// TwinCAT 3 PLC project Main
// ProgramVersion: 3.1.4024.0
// libraries:
//   Tc2_Standard, * (Beckhoff Automation GmbH)
//   Tc2_System, * (Beckhoff Automation GmbH)
//   Tc3_Module, * (Beckhoff Automation GmbH)
//   Tc3_Vision, * (Beckhoff Automation GmbH)
//   TcUnit, * (www.tcunit.org)
//   mobject-core,0.1.0,mobject
//   mobject-vision-nodepack,0.1.0,mobject
// project tree:
//   / PlcTask.TcTTO
//   POUs/ MAIN.TcPOU
//   Tests/Enums/ _ETcVn2dCodeSearchStrategy_TestSuite.TcPOU, _ETcVnAdaptiveThresholdMethod_TestSuite.TcPOU, _ETcVnBarcodeSearchDirection_TestSuite.TcPOU, _ETcVnBarcodeType_TestSuite.TcPOU, _ETcVnBlobCombination_TestSuite.TcPOU, _ETcVnBorderInterpolationMethod_TestSuite.TcPOU, _ETcVnColorSpaceTransform_TestSuite.TcPOU
// real-time tasks:
//   TASK PlcTask: cycle T#10ms, priority 20, ADS port 350

CONFIGURATION Main
    RESOURCE PLC ON TwinCAT3
        TASK PlcTask(INTERVAL := T#10ms, PRIORITY := 20);
        PROGRAM MAIN WITH PlcTask : MAIN;
    END_RESOURCE
END_CONFIGURATION

// ---- POUs/MAIN.TcPOU
PROGRAM MAIN
VAR
	
    // enums
    _ETcVn2dCodeSearchStrategy_TestSuite : _ETcVn2dCodeSearchStrategy_TestSuite;
    _ETcVnAdaptiveThresholdMethod_TestSuite : _ETcVnAdaptiveThresholdMethod_TestSuite;
    _ETcVnBarcodeSearchDirection_TestSuite : _ETcVnBarcodeSearchDirection_TestSuite;
    _ETcVnBarcodeType_TestSuite : _ETcVnBarcodeType_TestSuite;
    _ETcVnBlobCombination_TestSuite : _ETcVnBlobCombination_TestSuite;
    _ETcVnBorderInterpolationMethod_TestSuite : _ETcVnBorderInterpolationMethod_TestSuite;
    //_ETcVnCalibrationPattern_TestSuite : _ETcVnCalibrationPattern_TestSuite;
    //_ETcVnCalibrationPatternOrigin_TestSuite : _ETcVnCalibrationPatternOrigin_TestSuite;
    //_ETcVnCameraState_TestSuite : _ETcVnCameraState_TestSuite;
    //_ETcVnClusteringAlgorithm_TestSuite : _ETcVnClusteringAlgorithm_TestSuite;
    //_ETcVnColorMap_TestSuite : _ETcVnColorMap_TestSuite;
    //_ETcVnColorMapSize_TestSuite : _ETcVnColorMapSize_TestSuite;
    _ETcVnColorSpaceTransform_TestSuite : _ETcVnColorSpaceTransform_TestSuite;
    //_ETcVnColorTrainingMethod_TestSuite : _ETcVnColorTrainingMethod_TestSuite;
    //_ETcVnConnectedComponentsAlgorithm_TestSuite : _ETcVnConnectedComponentsAlgorithm_TestSuite;
    //_ETcVnContainerExportFormat_TestSuite : _ETcVnContainerExportFormat_TestSuite;
    //_ETcVnContourApproximationMethod_TestSuite : _ETcVnContourApproximationMethod_TestSuite;
    //_ETcVnContourRetrievalMode_TestSuite : _ETcVnContourRetrievalMode_TestSuite;
    //_ETcVnContoursMatchComparisonMethod_TestSuite : _ETcVnContoursMatchComparisonMethod_TestSuite;
    //_ETcVnDiffusivityTypeKAZE_TestSuite : _ETcVnDiffusivityTypeKAZE_TestSuite;
    //_ETcVnDistanceTransformationLabel_TestSuite : _ETcVnDistanceTransformationLabel_TestSuite;
    //_ETcVnDistanceTransformationMask_TestSuite : _ETcVnDistanceTransformationMask_TestSuite;
    //_ETcVnDistanceType_TestSuite : _ETcVnDistanceType_TestSuite;
    //_ETcVnDrawMatchesFlags_TestSuite : _ETcVnDrawMatchesFlags_TestSuite;
    //_ETcVnDrawShape_TestSuite : _ETcVnDrawShape_TestSuite;
    //_ETcVnEdgeDetectionAlgorithm_TestSuite : _ETcVnEdgeDetectionAlgorithm_TestSuite;
    //_ETcVnEdgeDirection_TestSuite : _ETcVnEdgeDirection_TestSuite;
    //_ETcVnElementType_TestSuite : _ETcVnElementType_TestSuite;
    //_ETcVnEstimationAlgorithm_TestSuite : _ETcVnEstimationAlgorithm_TestSuite;
    //_ETcVnExtremePointDirection_TestSuite : _ETcVnExtremePointDirection_TestSuite;
    //_ETcVnFeatureDescriptorTypeAKAZE_TestSuite : _ETcVnFeatureDescriptorTypeAKAZE_TestSuite;
    //_ETcVnFeatureScalingType_TestSuite : _ETcVnFeatureScalingType_TestSuite;
    //_ETcVnFeatureScoreTypeORB_TestSuite : _ETcVnFeatureScoreTypeORB_TestSuite;
    //_ETcVnFilterDirection_TestSuite : _ETcVnFilterDirection_TestSuite;
    //_ETcVnFlipAxis_TestSuite : _ETcVnFlipAxis_TestSuite;
    //_ETcVnFontType_TestSuite : _ETcVnFontType_TestSuite;
    //_ETcVnHoughMethod_TestSuite : _ETcVnHoughMethod_TestSuite;
    //_ETcVnInitializableFunction_TestSuite : _ETcVnInitializableFunction_TestSuite;
    //_ETcVnInterpolationType_TestSuite : _ETcVnInterpolationType_TestSuite;
    //_ETcVnKeypointDetectionTypeAGAST_TestSuite : _ETcVnKeypointDetectionTypeAGAST_TestSuite;
    //_ETcVnKeypointDetectionTypeFAST_TestSuite : _ETcVnKeypointDetectionTypeFAST_TestSuite;
    //_ETcVnKnn_TestSuite : _ETcVnKnn_TestSuite;
    //_ETcVnLineType_TestSuite : _ETcVnLineType_TestSuite;
    //_ETcVnMorphologicalOperator_TestSuite : _ETcVnMorphologicalOperator_TestSuite;
    //_ETcVnNbc_TestSuite : _ETcVnNbc_TestSuite;
    //_ETcVnNormalizationType_TestSuite : _ETcVnNormalizationType_TestSuite;
    //_ETcVnOcrModelType_TestSuite : _ETcVnOcrModelType_TestSuite;
    //_ETcVnOcrOptions_TestSuite : _ETcVnOcrOptions_TestSuite;
    //_ETcVnOrientationMethod_TestSuite : _ETcVnOrientationMethod_TestSuite;
    //_ETcVnPaddingMode_TestSuite : _ETcVnPaddingMode_TestSuite;
    //_ETcVnPixelConnectivity_TestSuite : _ETcVnPixelConnectivity_TestSuite;
    //_ETcVnPixelEncoding_TestSuite : _ETcVnPixelEncoding_TestSuite;
    //_ETcVnPixelPackMode_TestSuite : _ETcVnPixelPackMode_TestSuite;
    //_ETcVnPrototypeClusterer_TestSuite : _ETcVnPrototypeClusterer_TestSuite;
    //_ETcVnRectangleIntersection_TestSuite : _ETcVnRectangleIntersection_TestSuite;
    //_ETcVnRotationAngle_TestSuite : _ETcVnRotationAngle_TestSuite;
    //_ETcVnRTrees_TestSuite : _ETcVnRTrees_TestSuite;
    //_ETcVnSignedNormalization_TestSuite : _ETcVnSignedNormalization_TestSuite;
    //_ETcVnSolvePnPMethod_TestSuite : _ETcVnSolvePnPMethod_TestSuite;
    //_ETcVnSta_TestSuite : _ETcVnSta_TestSuite;
    //_ETcVnStructuringElementShape_TestSuite : _ETcVnStructuringElementShape_TestSuite;
    //_ETcVnSvm_TestSuite : _ETcVnSvm_TestSuite;
    //_ETcVnSvmKernelType_TestSuite : _ETcVnSvmKernelType_TestSuite;
    //_ETcVnSvmSgdClassifierMarginType_TestSuite : _ETcVnSvmSgdClassifierMarginType_TestSuite;
    //_ETcVnSvmSgdClassifierType_TestSuite : _ETcVnSvmSgdClassifierType_TestSuite;
    //_ETcVnTemplateMatchMethod_TestSuite : _ETcVnTemplateMatchMethod_TestSuite;
    //_ETcVnThresholdType_TestSuite : _ETcVnThresholdType_TestSuite;
    //_ETcVnVectorCompareMethod_TestSuite : _ETcVnVectorCompareMethod_TestSuite;
    //_ETcVnWorldCoordinateSystem_TestSuite : _ETcVnWorldCoordinateSystem_TestSuite;
    //_ETcWatchdogAccumulationType_TestSuite : _ETcWatchdogAccumulationType_TestSuite;
    //_GEV_CAMERA_STATE_TestSuite : _GEV_CAMERA_STATE_TestSuite;
    
    //structs
	
END_VAR

END_PROGRAM

// ---- Tests/Enums/_ETcVn2dCodeSearchStrategy_TestSuite.TcPOU
FUNCTION_BLOCK _ETcVn2dCodeSearchStrategy_TestSuite EXTENDS TcUnit.FB_TestSuite
VAR
END_VAR

TestAddress();
TestClearReference();
TestClone();
TestTypeNameReturnsExpected();
TestIdentifierReturnsExpected();
TestMakeReferenceToFollowsReference();
TestMakeReferenceToUpdatesReference();
TestSize();
TestValueReturnsExpectedAfterInit();
TestValueReturnsExpectedAfterChange();
TestSerializeTypeWith();
TestSerializeWith();
TestTryDeserializeFrom();
TestTryMakeReferenceToFollowsReference();
TestTryMakeReferenceToUpdatesReference();

METHOD PUBLIC TestAddress
VAR
    _type : _ETcVn2dCodeSearchStrategy(ETcVn2dCodeSearchStrategy.TCVN_CSS_DEFAULT);
    notExpected : PVOID := 0;
    actual : PVOID;
END_VAR
TEST('TestAddress');

actual := _type.Address;

AssertFalse(
    Condition := (notExpected = actual),
    Message := 'Type did not return a valid address.'
);

TEST_FINISHED();
END_METHOD

METHOD PUBLIC TestClearReference
VAR
    _type : _ETcVn2dCodeSearchStrategy(ETcVn2dCodeSearchStrategy.TCVN_CSS_DEFAULT);
	target : ETcVn2dCodeSearchStrategy := ETcVn2dCodeSearchStrategy.TCVN_CSS_DEFAULT;
    expected : ETcVn2dCodeSearchStrategy := ETcVn2dCodeSearchStrategy.TCVN_CSS_DEFAULT;
    actual : ETcVn2dCodeSearchStrategy;
END_VAR
TEST('TestClearReference');

_type.MakeReferenceTo(target);
_type.ClearReference();
target := ETcVn2dCodeSearchStrategy.TCVN_CSS_FIRST_FLIPPED;

actual := _type.Value;

AssertEquals(
    Expected := expected,
    Actual := actual,
    Message := 'Value continued to follow target.'
);

TEST_FINISHED();
END_METHOD

METHOD PUBLIC TestClone
VAR
    _type : _ETcVn2dCodeSearchStrategy(ETcVn2dCodeSearchStrategy.TCVN_CSS_DEFAULT);
	clone : I_Datatype;
	isValidClone : BOOL;
	compareResult : DINT;
END_VAR
TEST('TestClone');

clone := _type.Clone();

isValidClone := clone <> 0;

IF isValidClone THEN
	compareResult := memcmp(_type.Address, clone.Address, clone.Size);
END_IF

AssertTrue(
	Condition := isValidClone,
	Message := 'Clone did not produce a clone'
);

AssertEquals_DINT(
	Expected := 0,
    Actual := compareResult,
    Message := 'Clone did not return a valid clone.'
);

clone.Dispose();

TEST_FINISHED();
END_METHOD

METHOD PUBLIC TestIdentifierReturnsExpected
VAR
    _type : _ETcVn2dCodeSearchStrategy(ETcVn2dCodeSearchStrategy.TCVN_CSS_DEFAULT);
    expected : STRING := 'ETcVn2dCodeSearchStrategy';
    actual : STRING;
END_VAR
TEST('TestIdentifierReturnsExpected');

actual := _type.Identifier;

AssertEquals_STRING(
    Expected := expected,
    Actual := actual,
    Message := 'Type did not return correct iec type.'
);

TEST_FINISHED();
END_METHOD

METHOD PUBLIC TestMakeReferenceToFollowsReference
VAR
    _type : _ETcVn2dCodeSearchStrategy(ETcVn2dCodeSearchStrategy.TCVN_CSS_DEFAULT);
	target : ETcVn2dCodeSearchStrategy := ETcVn2dCodeSearchStrategy.TCVN_CSS_DEFAULT;
    expected : ETcVn2dCodeSearchStrategy := ETcVn2dCodeSearchStrategy.TCVN_CSS_FIRST_FLIPPED;
    actual : ETcVn2dCodeSearchStrategy;
END_VAR
TEST('TestMakeReferenceToFollowsReference');

_type.MakeReferenceTo(target);
target := ETcVn2dCodeSearchStrategy.TCVN_CSS_FIRST_FLIPPED;

actual := _type.Value;

AssertEquals(
    Expected := expected,
    Actual := actual,
    Message := 'Value did not follow target change.'
);

TEST_FINISHED();
END_METHOD

METHOD PUBLIC TestMakeReferenceToUpdatesReference
VAR
    _type : _ETcVn2dCodeSearchStrategy(ETcVn2dCodeSearchStrategy.TCVN_CSS_DEFAULT);
	target : ETcVn2dCodeSearchStrategy := ETcVn2dCodeSearchStrategy.TCVN_CSS_DEFAULT;
    expected : ETcVn2dCodeSearchStrategy := ETcVn2dCodeSearchStrategy.TCVN_CSS_FIRST_FLIPPED;
    actual : ETcVn2dCodeSearchStrategy;
END_VAR
TEST('TestMakeReferenceToUpdatesReference');

_type.MakeReferenceTo(target);
_type.Value := ETcVn2dCodeSearchStrategy.TCVN_CSS_FIRST_FLIPPED;

actual := target;

AssertEquals(
    Expected := expected,
    Actual := actual,
    Message := 'Value did not update target.'
);

TEST_FINISHED();
END_METHOD

METHOD PUBLIC TestSerializeTypeWith
VAR
    _type : _ETcVn2dCodeSearchStrategy(ETcVn2dCodeSearchStrategy.TCVN_CSS_DEFAULT);
    serializer : JsonSerializer;
    expected : STRING(500) := '{"typeName":"ENUM","identifier":"ETcVn2dCodeSearchStrategy","enumerations":["TCVN_CSS_DEFAULT","TCVN_CSS_FIRST_FLIPPED","TCVN_CSS_FIRST_INVERTED","TCVN_CSS_FIRST_NOT_FLIPPED","TCVN_CSS_FIRST_NOT_INVERTED","TCVN_CSS_ONLY_FLIPPED","TCVN_CSS_ONLY_INVERTED","TCVN_CSS_ONLY_NOT_FLIPPED","TCVN_CSS_ONLY_NOT_INVERTED"],"baseType":{"typeName":"UDINT","minValue":0,"maxValue":4294967295,"isSigned":false,"isFloat":false}}';
    actual : STRING(500);
END_VAR
TEST('TestSerializeTypeWith');

serializer.Reset();
_type.SerializeTypeWith(serializer);
serializer.TryGetSerializedData(ADR(actual), SIZEOF(actual));

AssertEquals_STRING(
    Expected := expected,
    Actual := actual,
    Message := 'Serialization of type did not return correct string.'
);

TEST_FINISHED();
END_METHOD

METHOD PUBLIC TestSerializeWith
VAR
    _type : _ETcVn2dCodeSearchStrategy(ETcVn2dCodeSearchStrategy.TCVN_CSS_DEFAULT);
    serializer : JsonSerializer;
    expected : STRING := '"TCVN_CSS_DEFAULT"';
    actual : STRING(500);
END_VAR
TEST('TestSerializeWith');

serializer.Reset();
_type.SerializeWith(serializer);
serializer.TryGetSerializedData(ADR(actual), SIZEOF(actual));

AssertEquals_STRING(
    Expected := expected,
    Actual := actual,
    Message := 'Serialization of type data did not return correct string.'
);

TEST_FINISHED();
END_METHOD

METHOD PUBLIC TestSize
VAR
    _type : _ETcVn2dCodeSearchStrategy(ETcVn2dCodeSearchStrategy.TCVN_CSS_DEFAULT);
    expected : UDINT := SIZEOF(ETcVn2dCodeSearchStrategy);
    actual : UDINT;
END_VAR
TEST('TestSize');

actual := _type.Size;

AssertEquals_UDINT(
    Expected := Expected,
    Actual := actual,
    Message := 'Type did not return the correct size.'
);

TEST_FINISHED();
END_METHOD

METHOD PUBLIC TestTryDeserializeFrom
VAR
    deserializer : JsonDeserializer;
    feedback : DeserializerFeedback;
    json : STRING := '"TCVN_CSS_DEFAULT"';
    _type : _ETcVn2dCodeSearchStrategy(ETcVn2dCodeSearchStrategy.TCVN_CSS_DEFAULT);
    expected : ETcVn2dCodeSearchStrategy := ETcVn2dCodeSearchStrategy.TCVN_CSS_DEFAULT;
    actual : ETcVn2dCodeSearchStrategy;
 END_VAR
TEST('TestTryDeserializeFrom');

deserializer.Reset();
deserializer.TryLoad(json);
_type.TryDeserializeFrom(Deserializer, Feedback);

actual := _type.Value;

AssertEquals(
    Expected := expected,
    Actual := actual,
    Message := 'Type did not deserialize correctly.'
);

TEST_FINISHED();
END_METHOD

METHOD PUBLIC TestTryMakeReferenceToFollowsReference
VAR
    _type : _ETcVn2dCodeSearchStrategy(ETcVn2dCodeSearchStrategy.TCVN_CSS_DEFAULT);
	target : _ETcVn2dCodeSearchStrategy(ETcVn2dCodeSearchStrategy.TCVN_CSS_DEFAULT);
    expected : ETcVn2dCodeSearchStrategy := ETcVn2dCodeSearchStrategy.TCVN_CSS_FIRST_FLIPPED;
    actual : ETcVn2dCodeSearchStrategy;
END_VAR
TEST('TestTryMakeReferenceToFollowsReference');

_type.TryMakeReferenceTo(target);
target.Value := ETcVn2dCodeSearchStrategy.TCVN_CSS_FIRST_FLIPPED;

actual := _type.Value;

AssertEquals(
    Expected := expected,
    Actual := actual,
    Message := 'Value did not follow target change.'
);

TEST_FINISHED();
END_METHOD

METHOD PUBLIC TestTryMakeReferenceToUpdatesReference
VAR
    _type : _ETcVn2dCodeSearchStrategy(ETcVn2dCodeSearchStrategy.TCVN_CSS_DEFAULT);
	target : _ETcVn2dCodeSearchStrategy(ETcVn2dCodeSearchStrategy.TCVN_CSS_DEFAULT);
    expected : ETcVn2dCodeSearchStrategy := ETcVn2dCodeSearchStrategy.TCVN_CSS_FIRST_FLIPPED;
    actual : ETcVn2dCodeSearchStrategy;
END_VAR
TEST('TestTryMakeReferenceToUpdatesReference');

_type.TryMakeReferenceTo(target);
_type.Value := ETcVn2dCodeSearchStrategy.TCVN_CSS_FIRST_FLIPPED;

actual := target.Value;

AssertEquals(
    Expected := expected,
    Actual := actual,
    Message := 'Value did not update target.'
);

TEST_FINISHED();
END_METHOD

METHOD PUBLIC TestTypeNameReturnsExpected
VAR
    _type : _ETcVn2dCodeSearchStrategy(ETcVn2dCodeSearchStrategy.TCVN_CSS_DEFAULT);
    expected : STRING := 'ENUM';
    actual : STRING;
END_VAR
TEST('TestTypeNameReturnsExpected');

actual := _type.TypeName;

AssertEquals_STRING(
    Expected := expected,
    Actual := actual,
    Message := 'Type did not return correct iec type.'
);

TEST_FINISHED();
END_METHOD

METHOD PUBLIC TestValueReturnsExpectedAfterChange
VAR
    _type : _ETcVn2dCodeSearchStrategy(ETcVn2dCodeSearchStrategy.TCVN_CSS_DEFAULT);
    expected : ETcVn2dCodeSearchStrategy := ETcVn2dCodeSearchStrategy.TCVN_CSS_FIRST_FLIPPED;
    actual : ETcVn2dCodeSearchStrategy;
END_VAR
TEST('TestValueReturnsExpectedAfterChange');

_type.Value := ETcVn2dCodeSearchStrategy.TCVN_CSS_FIRST_FLIPPED;

actual := _type.Value;

AssertEquals(
    Expected := expected,
    Actual := actual,
    Message := 'Expected value not returned after change.'
);

TEST_FINISHED();
END_METHOD

METHOD PUBLIC TestValueReturnsExpectedAfterInit
VAR
    _type : _ETcVn2dCodeSearchStrategy(ETcVn2dCodeSearchStrategy.TCVN_CSS_DEFAULT);
    expected : ETcVn2dCodeSearchStrategy := ETcVn2dCodeSearchStrategy.TCVN_CSS_DEFAULT;
    actual : ETcVn2dCodeSearchStrategy;
END_VAR
TEST('TestValueReturnsExpectedAfterInit');

actual := _type.Value;

AssertEquals(
    Expected := expected,
    Actual := actual,
    Message := 'Expected value not returned after Init.'
);

TEST_FINISHED();
END_METHOD

END_FUNCTION_BLOCK

// ---- Tests/Enums/_ETcVnAdaptiveThresholdMethod_TestSuite.TcPOU
FUNCTION_BLOCK _ETcVnAdaptiveThresholdMethod_TestSuite EXTENDS TcUnit.FB_TestSuite
VAR
END_VAR

TestAddress();
TestClearReference();
TestClone();
TestTypeNameReturnsExpected();
TestIdentifierReturnsExpected();
TestMakeReferenceToFollowsReference();
TestMakeReferenceToUpdatesReference();
TestSize();
TestValueReturnsExpectedAfterInit();
TestValueReturnsExpectedAfterChange();
TestSerializeTypeWith();
TestSerializeWith();
TestTryDeserializeFrom();
TestTryMakeReferenceToFollowsReference();
TestTryMakeReferenceToUpdatesReference();

METHOD PUBLIC TestAddress
VAR
    _type : _ETcVnAdaptiveThresholdMethod(ETcVnAdaptiveThresholdMethod.TCVN_ATM_MEAN);
    notExpected : PVOID := 0;
    actual : PVOID;
END_VAR
TEST('TestAddress');

actual := _type.Address;

AssertFalse(
    Condition := (notExpected = actual),
    Message := 'Type did not return a valid address.'
);

TEST_FINISHED();
END_METHOD

METHOD PUBLIC TestClearReference
VAR
    _type : _ETcVnAdaptiveThresholdMethod(ETcVnAdaptiveThresholdMethod.TCVN_ATM_MEAN);
	target : ETcVnAdaptiveThresholdMethod := ETcVnAdaptiveThresholdMethod.TCVN_ATM_MEAN;
    expected : ETcVnAdaptiveThresholdMethod := ETcVnAdaptiveThresholdMethod.TCVN_ATM_MEAN;
    actual : ETcVnAdaptiveThresholdMethod;
END_VAR
TEST('TestClearReference');

_type.MakeReferenceTo(target);
_type.ClearReference();
target := ETcVnAdaptiveThresholdMethod.TCVN_ATM_GAUSSIAN;

actual := _type.Value;

AssertEquals(
    Expected := expected,
    Actual := actual,
    Message := 'Value continued to follow target.'
);

TEST_FINISHED();
END_METHOD

METHOD PUBLIC TestClone
VAR
    _type : _ETcVnAdaptiveThresholdMethod(ETcVnAdaptiveThresholdMethod.TCVN_ATM_MEAN);
	clone : I_Datatype;
	isValidClone : BOOL;
	compareResult : DINT;
END_VAR
TEST('TestClone');

clone := _type.Clone();

isValidClone := clone <> 0;

IF isValidClone THEN
	compareResult := memcmp(_type.Address, clone.Address, clone.Size);
END_IF

AssertTrue(
	Condition := isValidClone,
	Message := 'Clone did not produce a clone'
);

AssertEquals_DINT(
	Expected := 0,
    Actual := compareResult,
    Message := 'Clone did not return a valid clone.'
);

clone.Dispose();

TEST_FINISHED();
END_METHOD

METHOD PUBLIC TestIdentifierReturnsExpected
VAR
    _type : _ETcVnAdaptiveThresholdMethod(ETcVnAdaptiveThresholdMethod.TCVN_ATM_MEAN);
    expected : STRING := 'ETcVnAdaptiveThresholdMethod';
    actual : STRING;
END_VAR
TEST('TestIdentifierReturnsExpected');

actual := _type.Identifier;

AssertEquals_STRING(
    Expected := expected,
    Actual := actual,
    Message := 'Type did not return correct iec type.'
);

TEST_FINISHED();
END_METHOD

METHOD PUBLIC TestMakeReferenceToFollowsReference
VAR
    _type : _ETcVnAdaptiveThresholdMethod(ETcVnAdaptiveThresholdMethod.TCVN_ATM_MEAN);
	target : ETcVnAdaptiveThresholdMethod := ETcVnAdaptiveThresholdMethod.TCVN_ATM_MEAN;
    expected : ETcVnAdaptiveThresholdMethod := ETcVnAdaptiveThresholdMethod.TCVN_ATM_GAUSSIAN;
    actual : ETcVnAdaptiveThresholdMethod;
END_VAR
TEST('TestMakeReferenceToFollowsReference');

_type.MakeReferenceTo(target);
target := ETcVnAdaptiveThresholdMethod.TCVN_ATM_GAUSSIAN;

actual := _type.Value;

AssertEquals(
    Expected := expected,
    Actual := actual,
    Message := 'Value did not follow target change.'
);

TEST_FINISHED();
END_METHOD

METHOD PUBLIC TestMakeReferenceToUpdatesReference
VAR
    _type : _ETcVnAdaptiveThresholdMethod(ETcVnAdaptiveThresholdMethod.TCVN_ATM_MEAN);
	target : ETcVnAdaptiveThresholdMethod := ETcVnAdaptiveThresholdMethod.TCVN_ATM_MEAN;
    expected : ETcVnAdaptiveThresholdMethod := ETcVnAdaptiveThresholdMethod.TCVN_ATM_GAUSSIAN;
    actual : ETcVnAdaptiveThresholdMethod;
END_VAR
TEST('TestMakeReferenceToUpdatesReference');

_type.MakeReferenceTo(target);
_type.Value := ETcVnAdaptiveThresholdMethod.TCVN_ATM_GAUSSIAN;

actual := target;

AssertEquals(
    Expected := expected,
    Actual := actual,
    Message := 'Value did not update target.'
);

TEST_FINISHED();
END_METHOD

METHOD PUBLIC TestSerializeTypeWith
VAR
    _type : _ETcVnAdaptiveThresholdMethod(ETcVnAdaptiveThresholdMethod.TCVN_ATM_MEAN);
    serializer : JsonSerializer;
    expected : STRING(500) := '{"typeName":"ENUM","identifier":"ETcVnAdaptiveThresholdMethod","enumerations":["TCVN_ATM_MEAN","TCVN_ATM_GAUSSIAN"],"baseType":{"typeName":"DINT","minValue":-2147483648,"maxValue":2147483647,"isSigned":true,"isFloat":false}}'; 
    actual : STRING(500);
END_VAR
TEST('TestSerializeTypeWith');

serializer.Reset();
_type.SerializeTypeWith(serializer);
serializer.TryGetSerializedData(ADR(actual), SIZEOF(actual));

AssertEquals_STRING(
    Expected := expected,
    Actual := actual,
    Message := 'Serialization of type did not return correct string.'
);

TEST_FINISHED();
END_METHOD

METHOD PUBLIC TestSerializeWith
VAR
    _type : _ETcVnAdaptiveThresholdMethod(ETcVnAdaptiveThresholdMethod.TCVN_ATM_MEAN);
    serializer : JsonSerializer;
    expected : STRING := '"TCVN_ATM_MEAN"';
    actual : STRING(500);
END_VAR
TEST('TestSerializeWith');

serializer.Reset();
_type.SerializeWith(serializer);
serializer.TryGetSerializedData(ADR(actual), SIZEOF(actual));

AssertEquals_STRING(
    Expected := expected,
    Actual := actual,
    Message := 'Serialization of type data did not return correct string.'
);

TEST_FINISHED();
END_METHOD

METHOD PUBLIC TestSize
VAR
    _type : _ETcVnAdaptiveThresholdMethod(ETcVnAdaptiveThresholdMethod.TCVN_ATM_MEAN);
    expected : UDINT := SIZEOF(ETcVnAdaptiveThresholdMethod);
    actual : UDINT;
END_VAR
TEST('TestSize');

actual := _type.Size;

AssertEquals_UDINT(
    Expected := Expected,
    Actual := actual,
    Message := 'Type did not return the correct size.'
);

TEST_FINISHED();
END_METHOD

METHOD PUBLIC TestTryDeserializeFrom
VAR
    deserializer : JsonDeserializer;
    feedback : DeserializerFeedback;
    json : STRING := '"TCVN_ATM_MEAN"';
    _type : _ETcVnAdaptiveThresholdMethod(ETcVnAdaptiveThresholdMethod.TCVN_ATM_MEAN);
    expected : ETcVnAdaptiveThresholdMethod := ETcVnAdaptiveThresholdMethod.TCVN_ATM_MEAN;
    actual : ETcVnAdaptiveThresholdMethod;
 END_VAR
TEST('TestTryDeserializeFrom');

deserializer.Reset();
deserializer.TryLoad(json);
_type.TryDeserializeFrom(Deserializer, Feedback);

actual := _type.Value;

AssertEquals(
    Expected := expected,
    Actual := actual,
    Message := 'Type did not deserialize correctly.'
);

TEST_FINISHED();
END_METHOD

METHOD PUBLIC TestTryMakeReferenceToFollowsReference
VAR
    _type : _ETcVnAdaptiveThresholdMethod(ETcVnAdaptiveThresholdMethod.TCVN_ATM_MEAN);
	target : _ETcVnAdaptiveThresholdMethod(ETcVnAdaptiveThresholdMethod.TCVN_ATM_MEAN);
    expected : ETcVnAdaptiveThresholdMethod := ETcVnAdaptiveThresholdMethod.TCVN_ATM_GAUSSIAN;
    actual : ETcVnAdaptiveThresholdMethod;
END_VAR
TEST('TestTryMakeReferenceToFollowsReference');

_type.TryMakeReferenceTo(target);
target.Value := ETcVnAdaptiveThresholdMethod.TCVN_ATM_GAUSSIAN;

actual := _type.Value;

AssertEquals(
    Expected := expected,
    Actual := actual,
    Message := 'Value did not follow target change.'
);

TEST_FINISHED();
END_METHOD

METHOD PUBLIC TestTryMakeReferenceToUpdatesReference
VAR
    _type : _ETcVnAdaptiveThresholdMethod(ETcVnAdaptiveThresholdMethod.TCVN_ATM_MEAN);
	target : _ETcVnAdaptiveThresholdMethod(ETcVnAdaptiveThresholdMethod.TCVN_ATM_MEAN);
    expected : ETcVnAdaptiveThresholdMethod := ETcVnAdaptiveThresholdMethod.TCVN_ATM_GAUSSIAN;
    actual : ETcVnAdaptiveThresholdMethod;
END_VAR
TEST('TestTryMakeReferenceToUpdatesReference');

_type.TryMakeReferenceTo(target);
_type.Value := ETcVnAdaptiveThresholdMethod.TCVN_ATM_GAUSSIAN;

actual := target.Value;

AssertEquals(
    Expected := expected,
    Actual := actual,
    Message := 'Value did not update target.'
);

TEST_FINISHED();
END_METHOD

METHOD PUBLIC TestTypeNameReturnsExpected
VAR
    _type : _ETcVnAdaptiveThresholdMethod(ETcVnAdaptiveThresholdMethod.TCVN_ATM_MEAN);
    expected : STRING := 'ENUM';
    actual : STRING;
END_VAR
TEST('TestTypeNameReturnsExpected');

actual := _type.TypeName;

AssertEquals_STRING(
    Expected := expected,
    Actual := actual,
    Message := 'Type did not return correct iec type.'
);

TEST_FINISHED();
END_METHOD

METHOD PUBLIC TestValueReturnsExpectedAfterChange
VAR
    _type : _ETcVnAdaptiveThresholdMethod(ETcVnAdaptiveThresholdMethod.TCVN_ATM_MEAN);
    expected : ETcVnAdaptiveThresholdMethod := ETcVnAdaptiveThresholdMethod.TCVN_ATM_GAUSSIAN;
    actual : ETcVnAdaptiveThresholdMethod;
END_VAR
TEST('TestValueReturnsExpectedAfterChange');

_type.Value := ETcVnAdaptiveThresholdMethod.TCVN_ATM_GAUSSIAN;

actual := _type.Value;

AssertEquals(
    Expected := expected,
    Actual := actual,
    Message := 'Expected value not returned after change.'
);

TEST_FINISHED();
END_METHOD

METHOD PUBLIC TestValueReturnsExpectedAfterInit
VAR
    _type : _ETcVnAdaptiveThresholdMethod(ETcVnAdaptiveThresholdMethod.TCVN_ATM_MEAN);
    expected : ETcVnAdaptiveThresholdMethod := ETcVnAdaptiveThresholdMethod.TCVN_ATM_MEAN;
    actual : ETcVnAdaptiveThresholdMethod;
END_VAR
TEST('TestValueReturnsExpectedAfterInit');

actual := _type.Value;

AssertEquals(
    Expected := expected,
    Actual := actual,
    Message := 'Expected value not returned after Init.'
);

TEST_FINISHED();
END_METHOD

END_FUNCTION_BLOCK

// ---- Tests/Enums/_ETcVnBarcodeSearchDirection_TestSuite.TcPOU
FUNCTION_BLOCK _ETcVnBarcodeSearchDirection_TestSuite EXTENDS TcUnit.FB_TestSuite
VAR
END_VAR

TestAddress();
TestClearReference();
TestClone();
TestTypeNameReturnsExpected();
TestIdentifierReturnsExpected();
TestMakeReferenceToFollowsReference();
TestMakeReferenceToUpdatesReference();
TestSize();
TestValueReturnsExpectedAfterInit();
TestValueReturnsExpectedAfterChange();
TestSerializeTypeWith();
TestSerializeWith();
TestTryDeserializeFrom();
TestTryMakeReferenceToFollowsReference();
TestTryMakeReferenceToUpdatesReference();

METHOD PUBLIC TestAddress
VAR
    _type : _ETcVnBarcodeSearchDirection(ETcVnBarcodeSearchDirection.TCVN_BSD_ANY);
    notExpected : PVOID := 0;
    actual : PVOID;
END_VAR
TEST('TestAddress');

actual := _type.Address;

AssertFalse(
    Condition := (notExpected = actual),
    Message := 'Type did not return a valid address.'
);

TEST_FINISHED();
END_METHOD

METHOD PUBLIC TestClearReference
VAR
    _type : _ETcVnBarcodeSearchDirection(ETcVnBarcodeSearchDirection.TCVN_BSD_ANY);
	target : ETcVnBarcodeSearchDirection := ETcVnBarcodeSearchDirection.TCVN_BSD_ANY;
    expected : ETcVnBarcodeSearchDirection := ETcVnBarcodeSearchDirection.TCVN_BSD_ANY;
    actual : ETcVnBarcodeSearchDirection;
END_VAR
TEST('TestClearReference');

_type.MakeReferenceTo(target);
_type.ClearReference();
target := ETcVnBarcodeSearchDirection.TCVN_BSD_HORIZONTAL;

actual := _type.Value;

AssertEquals(
    Expected := expected,
    Actual := actual,
    Message := 'Value continued to follow target.'
);

TEST_FINISHED();
END_METHOD

METHOD PUBLIC TestClone
VAR
    _type : _ETcVnBarcodeSearchDirection(ETcVnBarcodeSearchDirection.TCVN_BSD_ANY);
	clone : I_Datatype;
	isValidClone : BOOL;
	compareResult : DINT;
END_VAR
TEST('TestClone');

clone := _type.Clone();

isValidClone := clone <> 0;

IF isValidClone THEN
	compareResult := memcmp(_type.Address, clone.Address, clone.Size);
END_IF

AssertTrue(
	Condition := isValidClone,
	Message := 'Clone did not produce a clone'
);

AssertEquals_DINT(
	Expected := 0,
    Actual := compareResult,
    Message := 'Clone did not return a valid clone.'
);

clone.Dispose();

TEST_FINISHED();
END_METHOD

METHOD PUBLIC TestIdentifierReturnsExpected
VAR
    _type : _ETcVnBarcodeSearchDirection(ETcVnBarcodeSearchDirection.TCVN_BSD_ANY);
    expected : STRING := 'ETcVnBarcodeSearchDirection';
    actual : STRING;
END_VAR
TEST('TestIdentifierReturnsExpected');

actual := _type.Identifier;

AssertEquals_STRING(
    Expected := expected,
    Actual := actual,
    Message := 'Type did not return correct iec type.'
);

TEST_FINISHED();
END_METHOD

METHOD PUBLIC TestMakeReferenceToFollowsReference
VAR
    _type : _ETcVnBarcodeSearchDirection(ETcVnBarcodeSearchDirection.TCVN_BSD_ANY);
	target : ETcVnBarcodeSearchDirection := ETcVnBarcodeSearchDirection.TCVN_BSD_ANY;
    expected : ETcVnBarcodeSearchDirection := ETcVnBarcodeSearchDirection.TCVN_BSD_HORIZONTAL;
    actual : ETcVnBarcodeSearchDirection;
END_VAR
TEST('TestMakeReferenceToFollowsReference');

_type.MakeReferenceTo(target);
target := ETcVnBarcodeSearchDirection.TCVN_BSD_HORIZONTAL;

actual := _type.Value;

AssertEquals(
    Expected := expected,
    Actual := actual,
    Message := 'Value did not follow target change.'
);

TEST_FINISHED();
END_METHOD

METHOD PUBLIC TestMakeReferenceToUpdatesReference
VAR
    _type : _ETcVnBarcodeSearchDirection(ETcVnBarcodeSearchDirection.TCVN_BSD_ANY);
	target : ETcVnBarcodeSearchDirection := ETcVnBarcodeSearchDirection.TCVN_BSD_ANY;
    expected : ETcVnBarcodeSearchDirection := ETcVnBarcodeSearchDirection.TCVN_BSD_HORIZONTAL;
    actual : ETcVnBarcodeSearchDirection;
END_VAR
TEST('TestMakeReferenceToUpdatesReference');

_type.MakeReferenceTo(target);
_type.Value := ETcVnBarcodeSearchDirection.TCVN_BSD_HORIZONTAL;

actual := target;

AssertEquals(
    Expected := expected,
    Actual := actual,
    Message := 'Value did not update target.'
);

TEST_FINISHED();
END_METHOD

METHOD PUBLIC TestSerializeTypeWith
VAR
    _type : _ETcVnBarcodeSearchDirection(ETcVnBarcodeSearchDirection.TCVN_BSD_ANY);
    serializer : JsonSerializer;
    expected : STRING(500) := '{"typeName":"ENUM","identifier":"ETcVnBarcodeSearchDirection","enumerations":["TCVN_BSD_ANY","TCVN_BSD_HORIZONTAL","TCVN_BSD_VERTICAL"],"baseType":{"typeName":"UDINT","minValue":0,"maxValue":4294967295,"isSigned":false,"isFloat":false}}'; 
    actual : STRING(500);
END_VAR
TEST('TestSerializeTypeWith');

serializer.Reset();
_type.SerializeTypeWith(serializer);
serializer.TryGetSerializedData(ADR(actual), SIZEOF(actual));

AssertEquals_STRING(
    Expected := expected,
    Actual := actual,
    Message := 'Serialization of type did not return correct string.'
);

TEST_FINISHED();
END_METHOD

METHOD PUBLIC TestSerializeWith
VAR
    _type : _ETcVnBarcodeSearchDirection(ETcVnBarcodeSearchDirection.TCVN_BSD_ANY);
    serializer : JsonSerializer;
    expected : STRING := '"TCVN_BSD_ANY"';
    actual : STRING(500);
END_VAR
TEST('TestSerializeWith');

serializer.Reset();
_type.SerializeWith(serializer);
serializer.TryGetSerializedData(ADR(actual), SIZEOF(actual));

AssertEquals_STRING(
    Expected := expected,
    Actual := actual,
    Message := 'Serialization of type data did not return correct string.'
);

TEST_FINISHED();
END_METHOD

METHOD PUBLIC TestSize
VAR
    _type : _ETcVnBarcodeSearchDirection(ETcVnBarcodeSearchDirection.TCVN_BSD_ANY);
    expected : UDINT := SIZEOF(ETcVnBarcodeSearchDirection);
    actual : UDINT;
END_VAR
TEST('TestSize');

actual := _type.Size;

AssertEquals_UDINT(
    Expected := Expected,
    Actual := actual,
    Message := 'Type did not return the correct size.'
);

TEST_FINISHED();
END_METHOD

METHOD PUBLIC TestTryDeserializeFrom
VAR
    deserializer : JsonDeserializer;
    feedback : DeserializerFeedback;
    json : STRING := '"TCVN_BSD_ANY"';
    _type : _ETcVnBarcodeSearchDirection(ETcVnBarcodeSearchDirection.TCVN_BSD_ANY);
    expected : ETcVnBarcodeSearchDirection := ETcVnBarcodeSearchDirection.TCVN_BSD_ANY;
    actual : ETcVnBarcodeSearchDirection;
 END_VAR
TEST('TestTryDeserializeFrom');

deserializer.Reset();
deserializer.TryLoad(json);
_type.TryDeserializeFrom(Deserializer, Feedback);

actual := _type.Value;

AssertEquals(
    Expected := expected,
    Actual := actual,
    Message := 'Type did not deserialize correctly.'
);

TEST_FINISHED();
END_METHOD

METHOD PUBLIC TestTryMakeReferenceToFollowsReference
VAR
    _type : _ETcVnBarcodeSearchDirection(ETcVnBarcodeSearchDirection.TCVN_BSD_ANY);
	target : _ETcVnBarcodeSearchDirection(ETcVnBarcodeSearchDirection.TCVN_BSD_ANY);
    expected : ETcVnBarcodeSearchDirection := ETcVnBarcodeSearchDirection.TCVN_BSD_HORIZONTAL;
    actual : ETcVnBarcodeSearchDirection;
END_VAR
TEST('TestTryMakeReferenceToFollowsReference');

_type.TryMakeReferenceTo(target);
target.Value := ETcVnBarcodeSearchDirection.TCVN_BSD_HORIZONTAL;

actual := _type.Value;

AssertEquals(
    Expected := expected,
    Actual := actual,
    Message := 'Value did not follow target change.'
);

TEST_FINISHED();
END_METHOD

METHOD PUBLIC TestTryMakeReferenceToUpdatesReference
VAR
    _type : _ETcVnBarcodeSearchDirection(ETcVnBarcodeSearchDirection.TCVN_BSD_ANY);
	target : _ETcVnBarcodeSearchDirection(ETcVnBarcodeSearchDirection.TCVN_BSD_ANY);
    expected : ETcVnBarcodeSearchDirection := ETcVnBarcodeSearchDirection.TCVN_BSD_HORIZONTAL;
    actual : ETcVnBarcodeSearchDirection;
END_VAR
TEST('TestTryMakeReferenceToUpdatesReference');

_type.TryMakeReferenceTo(target);
_type.Value := ETcVnBarcodeSearchDirection.TCVN_BSD_HORIZONTAL;

actual := target.Value;

AssertEquals(
    Expected := expected,
    Actual := actual,
    Message := 'Value did not update target.'
);

TEST_FINISHED();
END_METHOD

METHOD PUBLIC TestTypeNameReturnsExpected
VAR
    _type : _ETcVnBarcodeSearchDirection(ETcVnBarcodeSearchDirection.TCVN_BSD_ANY);
    expected : STRING := 'ENUM';
    actual : STRING;
END_VAR
TEST('TestTypeNameReturnsExpected');

actual := _type.TypeName;

AssertEquals_STRING(
    Expected := expected,
    Actual := actual,
    Message := 'Type did not return correct iec type.'
);

TEST_FINISHED();
END_METHOD

METHOD PUBLIC TestValueReturnsExpectedAfterChange
VAR
    _type : _ETcVnBarcodeSearchDirection(ETcVnBarcodeSearchDirection.TCVN_BSD_ANY);
    expected : ETcVnBarcodeSearchDirection := ETcVnBarcodeSearchDirection.TCVN_BSD_HORIZONTAL;
    actual : ETcVnBarcodeSearchDirection;
END_VAR
TEST('TestValueReturnsExpectedAfterChange');

_type.Value := ETcVnBarcodeSearchDirection.TCVN_BSD_HORIZONTAL;

actual := _type.Value;

AssertEquals(
    Expected := expected,
    Actual := actual,
    Message := 'Expected value not returned after change.'
);

TEST_FINISHED();
END_METHOD

METHOD PUBLIC TestValueReturnsExpectedAfterInit
VAR
    _type : _ETcVnBarcodeSearchDirection(ETcVnBarcodeSearchDirection.TCVN_BSD_ANY);
    expected : ETcVnBarcodeSearchDirection := ETcVnBarcodeSearchDirection.TCVN_BSD_ANY;
    actual : ETcVnBarcodeSearchDirection;
END_VAR
TEST('TestValueReturnsExpectedAfterInit');

actual := _type.Value;

AssertEquals(
    Expected := expected,
    Actual := actual,
    Message := 'Expected value not returned after Init.'
);

TEST_FINISHED();
END_METHOD

END_FUNCTION_BLOCK

// ---- Tests/Enums/_ETcVnBarcodeType_TestSuite.TcPOU
FUNCTION_BLOCK _ETcVnBarcodeType_TestSuite EXTENDS TcUnit.FB_TestSuite
VAR
END_VAR

TestAddress();
TestClearReference();
TestClone();
TestTypeNameReturnsExpected();
TestIdentifierReturnsExpected();
TestMakeReferenceToFollowsReference();
TestMakeReferenceToUpdatesReference();
TestSize();
TestValueReturnsExpectedAfterInit();
TestValueReturnsExpectedAfterChange();
TestSerializeTypeWith();
TestSerializeWith();
TestTryDeserializeFrom();
TestTryMakeReferenceToFollowsReference();
TestTryMakeReferenceToUpdatesReference();

METHOD PUBLIC TestAddress
VAR
    _type : _ETcVnBarcodeType(ETcVnBarcodeType.TCVN_BT_CODABAR);
    notExpected : PVOID := 0;
    actual : PVOID;
END_VAR
TEST('TestAddress');

actual := _type.Address;

AssertFalse(
    Condition := (notExpected = actual),
    Message := 'Type did not return a valid address.'
);

TEST_FINISHED();
END_METHOD

METHOD PUBLIC TestClearReference
VAR
    _type : _ETcVnBarcodeType(ETcVnBarcodeType.TCVN_BT_CODABAR);
	target : ETcVnBarcodeType := ETcVnBarcodeType.TCVN_BT_CODABAR;
    expected : ETcVnBarcodeType := ETcVnBarcodeType.TCVN_BT_CODABAR;
    actual : ETcVnBarcodeType;
END_VAR
TEST('TestClearReference');

_type.MakeReferenceTo(target);
_type.ClearReference();
target := ETcVnBarcodeType.TCVN_BT_CODE39;

actual := _type.Value;

AssertEquals(
    Expected := expected,
    Actual := actual,
    Message := 'Value continued to follow target.'
);

TEST_FINISHED();
END_METHOD

METHOD PUBLIC TestClone
VAR
    _type : _ETcVnBarcodeType(ETcVnBarcodeType.TCVN_BT_CODABAR);
	clone : I_Datatype;
	isValidClone : BOOL;
	compareResult : DINT;
END_VAR
TEST('TestClone');

clone := _type.Clone();

isValidClone := clone <> 0;

IF isValidClone THEN
	compareResult := memcmp(_type.Address, clone.Address, clone.Size);
END_IF

AssertTrue(
	Condition := isValidClone,
	Message := 'Clone did not produce a clone'
);

AssertEquals_DINT(
	Expected := 0,
    Actual := compareResult,
    Message := 'Clone did not return a valid clone.'
);

clone.Dispose();

TEST_FINISHED();
END_METHOD

METHOD PUBLIC TestIdentifierReturnsExpected
VAR
    _type : _ETcVnBarcodeType(ETcVnBarcodeType.TCVN_BT_CODABAR);
    expected : STRING := 'ETcVnBarcodeType';
    actual : STRING;
END_VAR
TEST('TestIdentifierReturnsExpected');

actual := _type.Identifier;

AssertEquals_STRING(
    Expected := expected,
    Actual := actual,
    Message := 'Type did not return correct iec type.'
);

TEST_FINISHED();
END_METHOD

METHOD PUBLIC TestMakeReferenceToFollowsReference
VAR
    _type : _ETcVnBarcodeType(ETcVnBarcodeType.TCVN_BT_CODABAR);
	target : ETcVnBarcodeType := ETcVnBarcodeType.TCVN_BT_CODABAR;
    expected : ETcVnBarcodeType := ETcVnBarcodeType.TCVN_BT_CODE39;
    actual : ETcVnBarcodeType;
END_VAR
TEST('TestMakeReferenceToFollowsReference');

_type.MakeReferenceTo(target);
target := ETcVnBarcodeType.TCVN_BT_CODE39;

actual := _type.Value;

AssertEquals(
    Expected := expected,
    Actual := actual,
    Message := 'Value did not follow target change.'
);

TEST_FINISHED();
END_METHOD

METHOD PUBLIC TestMakeReferenceToUpdatesReference
VAR
    _type : _ETcVnBarcodeType(ETcVnBarcodeType.TCVN_BT_CODABAR);
	target : ETcVnBarcodeType := ETcVnBarcodeType.TCVN_BT_CODABAR;
    expected : ETcVnBarcodeType := ETcVnBarcodeType.TCVN_BT_CODE39;
    actual : ETcVnBarcodeType;
END_VAR
TEST('TestMakeReferenceToUpdatesReference');

_type.MakeReferenceTo(target);
_type.Value := ETcVnBarcodeType.TCVN_BT_CODE39;

actual := target;

AssertEquals(
    Expected := expected,
    Actual := actual,
    Message := 'Value did not update target.'
);

TEST_FINISHED();
END_METHOD

METHOD PUBLIC TestSerializeTypeWith
VAR
    _type : _ETcVnBarcodeType(ETcVnBarcodeType.TCVN_BT_CODABAR);
    serializer : JsonSerializer;
    expected : STRING(500) := '{"typeName":"ENUM","identifier":"ETcVnBarcodeType","enumerations":["TCVN_BT_CODABAR","TCVN_BT_CODE39","TCVN_BT_CODE93","TCVN_BT_CODE128","TCVN_BT_EAN8","TCVN_BT_EAN13","TCVN_BT_ITF","TCVN_BT_UPCA","TCVN_BT_UPCE","TCVN_BT_ANY","TCVN_BT_CODE39EXTENDED"],"baseType":{"typeName":"UDINT","minValue":0,"maxValue":4294967295,"isSigned":false,"isFloat":false}}'; 
    actual : STRING(500);
END_VAR
TEST('TestSerializeTypeWith');

serializer.Reset();
_type.SerializeTypeWith(serializer);
serializer.TryGetSerializedData(ADR(actual), SIZEOF(actual));

AssertEquals_STRING(
    Expected := expected,
    Actual := actual,
    Message := 'Serialization of type did not return correct string.'
);

TEST_FINISHED();
END_METHOD

METHOD PUBLIC TestSerializeWith
VAR
    _type : _ETcVnBarcodeType(ETcVnBarcodeType.TCVN_BT_CODABAR);
    serializer : JsonSerializer;
    expected : STRING := '"TCVN_BT_CODABAR"';
    actual : STRING(500);
END_VAR
TEST('TestSerializeWith');

serializer.Reset();
_type.SerializeWith(serializer);
serializer.TryGetSerializedData(ADR(actual), SIZEOF(actual));

AssertEquals_STRING(
    Expected := expected,
    Actual := actual,
    Message := 'Serialization of type data did not return correct string.'
);

TEST_FINISHED();
END_METHOD

METHOD PUBLIC TestSize
VAR
    _type : _ETcVnBarcodeType(ETcVnBarcodeType.TCVN_BT_CODABAR);
    expected : UDINT := SIZEOF(ETcVnBarcodeType);
    actual : UDINT;
END_VAR
TEST('TestSize');

actual := _type.Size;

AssertEquals_UDINT(
    Expected := Expected,
    Actual := actual,
    Message := 'Type did not return the correct size.'
);

TEST_FINISHED();
END_METHOD

METHOD PUBLIC TestTryDeserializeFrom
VAR
    deserializer : JsonDeserializer;
    feedback : DeserializerFeedback;
    json : STRING := '"TCVN_BT_CODABAR"';
    _type : _ETcVnBarcodeType(ETcVnBarcodeType.TCVN_BT_CODABAR);
    expected : ETcVnBarcodeType := ETcVnBarcodeType.TCVN_BT_CODABAR;
    actual : ETcVnBarcodeType;
 END_VAR
TEST('TestTryDeserializeFrom');

deserializer.Reset();
deserializer.TryLoad(json);
_type.TryDeserializeFrom(Deserializer, Feedback);

actual := _type.Value;

AssertEquals(
    Expected := expected,
    Actual := actual,
    Message := 'Type did not deserialize correctly.'
);

TEST_FINISHED();
END_METHOD

METHOD PUBLIC TestTryMakeReferenceToFollowsReference
VAR
    _type : _ETcVnBarcodeType(ETcVnBarcodeType.TCVN_BT_CODABAR);
	target : _ETcVnBarcodeType(ETcVnBarcodeType.TCVN_BT_CODABAR);
    expected : ETcVnBarcodeType := ETcVnBarcodeType.TCVN_BT_CODE39;
    actual : ETcVnBarcodeType;
END_VAR
TEST('TestTryMakeReferenceToFollowsReference');

_type.TryMakeReferenceTo(target);
target.Value := ETcVnBarcodeType.TCVN_BT_CODE39;

actual := _type.Value;

AssertEquals(
    Expected := expected,
    Actual := actual,
    Message := 'Value did not follow target change.'
);

TEST_FINISHED();
END_METHOD

METHOD PUBLIC TestTryMakeReferenceToUpdatesReference
VAR
    _type : _ETcVnBarcodeType(ETcVnBarcodeType.TCVN_BT_CODABAR);
	target : _ETcVnBarcodeType(ETcVnBarcodeType.TCVN_BT_CODABAR);
    expected : ETcVnBarcodeType := ETcVnBarcodeType.TCVN_BT_CODE39;
    actual : ETcVnBarcodeType;
END_VAR
TEST('TestTryMakeReferenceToUpdatesReference');

_type.TryMakeReferenceTo(target);
_type.Value := ETcVnBarcodeType.TCVN_BT_CODE39;

actual := target.Value;

AssertEquals(
    Expected := expected,
    Actual := actual,
    Message := 'Value did not update target.'
);

TEST_FINISHED();
END_METHOD

METHOD PUBLIC TestTypeNameReturnsExpected
VAR
    _type : _ETcVnBarcodeType(ETcVnBarcodeType.TCVN_BT_CODABAR);
    expected : STRING := 'ENUM';
    actual : STRING;
END_VAR
TEST('TestTypeNameReturnsExpected');

actual := _type.TypeName;

AssertEquals_STRING(
    Expected := expected,
    Actual := actual,
    Message := 'Type did not return correct iec type.'
);

TEST_FINISHED();
END_METHOD

METHOD PUBLIC TestValueReturnsExpectedAfterChange
VAR
    _type : _ETcVnBarcodeType(ETcVnBarcodeType.TCVN_BT_CODABAR);
    expected : ETcVnBarcodeType := ETcVnBarcodeType.TCVN_BT_CODE39;
    actual : ETcVnBarcodeType;
END_VAR
TEST('TestValueReturnsExpectedAfterChange');

_type.Value := ETcVnBarcodeType.TCVN_BT_CODE39;

actual := _type.Value;

AssertEquals(
    Expected := expected,
    Actual := actual,
    Message := 'Expected value not returned after change.'
);

TEST_FINISHED();
END_METHOD

METHOD PUBLIC TestValueReturnsExpectedAfterInit
VAR
    _type : _ETcVnBarcodeType(ETcVnBarcodeType.TCVN_BT_CODABAR);
    expected : ETcVnBarcodeType := ETcVnBarcodeType.TCVN_BT_CODABAR;
    actual : ETcVnBarcodeType;
END_VAR
TEST('TestValueReturnsExpectedAfterInit');

actual := _type.Value;

AssertEquals(
    Expected := expected,
    Actual := actual,
    Message := 'Expected value not returned after Init.'
);

TEST_FINISHED();
END_METHOD

END_FUNCTION_BLOCK

// ---- Tests/Enums/_ETcVnBlobCombination_TestSuite.TcPOU
FUNCTION_BLOCK _ETcVnBlobCombination_TestSuite EXTENDS TcUnit.FB_TestSuite
VAR
END_VAR

TestAddress();
TestClearReference();
TestClone();
TestTypeNameReturnsExpected();
TestIdentifierReturnsExpected();
TestMakeReferenceToFollowsReference();
TestMakeReferenceToUpdatesReference();
TestSize();
TestValueReturnsExpectedAfterInit();
TestValueReturnsExpectedAfterChange();
TestSerializeTypeWith();
TestSerializeWith();
TestTryDeserializeFrom();
TestTryMakeReferenceToFollowsReference();
TestTryMakeReferenceToUpdatesReference();

METHOD PUBLIC TestAddress
VAR
    _type : _ETcVnBlobCombination(ETcVnBlobCombination.TCVN_BC_SMALLEST);
    notExpected : PVOID := 0;
    actual : PVOID;
END_VAR
TEST('TestAddress');

actual := _type.Address;

AssertFalse(
    Condition := (notExpected = actual),
    Message := 'Type did not return a valid address.'
);

TEST_FINISHED();
END_METHOD

METHOD PUBLIC TestClearReference
VAR
    _type : _ETcVnBlobCombination(ETcVnBlobCombination.TCVN_BC_SMALLEST);
	target : ETcVnBlobCombination := ETcVnBlobCombination.TCVN_BC_SMALLEST;
    expected : ETcVnBlobCombination := ETcVnBlobCombination.TCVN_BC_SMALLEST;
    actual : ETcVnBlobCombination;
END_VAR
TEST('TestClearReference');

_type.MakeReferenceTo(target);
_type.ClearReference();
target := ETcVnBlobCombination.TCVN_BC_LARGEST;

actual := _type.Value;

AssertEquals(
    Expected := expected,
    Actual := actual,
    Message := 'Value continued to follow target.'
);

TEST_FINISHED();
END_METHOD

METHOD PUBLIC TestClone
VAR
    _type : _ETcVnBlobCombination(ETcVnBlobCombination.TCVN_BC_SMALLEST);
	clone : I_Datatype;
	isValidClone : BOOL;
	compareResult : DINT;
END_VAR
TEST('TestClone');

clone := _type.Clone();

isValidClone := clone <> 0;

IF isValidClone THEN
	compareResult := memcmp(_type.Address, clone.Address, clone.Size);
END_IF

AssertTrue(
	Condition := isValidClone,
	Message := 'Clone did not produce a clone'
);

AssertEquals_DINT(
	Expected := 0,
    Actual := compareResult,
    Message := 'Clone did not return a valid clone.'
);

clone.Dispose();

TEST_FINISHED();
END_METHOD

METHOD PUBLIC TestIdentifierReturnsExpected
VAR
    _type : _ETcVnBlobCombination(ETcVnBlobCombination.TCVN_BC_SMALLEST);
    expected : STRING := 'ETcVnBlobCombination';
    actual : STRING;
END_VAR
TEST('TestIdentifierReturnsExpected');

actual := _type.Identifier;

AssertEquals_STRING(
    Expected := expected,
    Actual := actual,
    Message := 'Type did not return correct iec type.'
);

TEST_FINISHED();
END_METHOD

METHOD PUBLIC TestMakeReferenceToFollowsReference
VAR
    _type : _ETcVnBlobCombination(ETcVnBlobCombination.TCVN_BC_SMALLEST);
	target : ETcVnBlobCombination := ETcVnBlobCombination.TCVN_BC_SMALLEST;
    expected : ETcVnBlobCombination := ETcVnBlobCombination.TCVN_BC_LARGEST;
    actual : ETcVnBlobCombination;
END_VAR
TEST('TestMakeReferenceToFollowsReference');

_type.MakeReferenceTo(target);
target := ETcVnBlobCombination.TCVN_BC_LARGEST;

actual := _type.Value;

AssertEquals(
    Expected := expected,
    Actual := actual,
    Message := 'Value did not follow target change.'
);

TEST_FINISHED();
END_METHOD

METHOD PUBLIC TestMakeReferenceToUpdatesReference
VAR
    _type : _ETcVnBlobCombination(ETcVnBlobCombination.TCVN_BC_SMALLEST);
	target : ETcVnBlobCombination := ETcVnBlobCombination.TCVN_BC_SMALLEST;
    expected : ETcVnBlobCombination := ETcVnBlobCombination.TCVN_BC_LARGEST;
    actual : ETcVnBlobCombination;
END_VAR
TEST('TestMakeReferenceToUpdatesReference');

_type.MakeReferenceTo(target);
_type.Value := ETcVnBlobCombination.TCVN_BC_LARGEST;

actual := target;

AssertEquals(
    Expected := expected,
    Actual := actual,
    Message := 'Value did not update target.'
);

TEST_FINISHED();
END_METHOD

METHOD PUBLIC TestSerializeTypeWith
VAR
    _type : _ETcVnBlobCombination(ETcVnBlobCombination.TCVN_BC_SMALLEST);
    serializer : JsonSerializer;
    expected : STRING(500) := '{"typeName":"ENUM","identifier":"ETcVnBlobCombination","enumerations":["TCVN_BC_SMALLEST","TCVN_BC_LARGEST","TCVN_BC_MIN_THRESHOLD","TCVN_BC_MAX_THRESHOLD","TCVN_BC_MEDIAN_THRESHOLD"],"baseType":{"typeName":"DINT","minValue":-2147483648,"maxValue":2147483647,"isSigned":true,"isFloat":false}}';
    actual : STRING(500);
END_VAR
TEST('TestSerializeTypeWith');

serializer.Reset();
_type.SerializeTypeWith(serializer);
serializer.TryGetSerializedData(ADR(actual), SIZEOF(actual));

AssertEquals_STRING(
    Expected := expected,
    Actual := actual,
    Message := 'Serialization of type did not return correct string.'
);

TEST_FINISHED();
END_METHOD

METHOD PUBLIC TestSerializeWith
VAR
    _type : _ETcVnBlobCombination(ETcVnBlobCombination.TCVN_BC_SMALLEST);
    serializer : JsonSerializer;
    expected : STRING := '"TCVN_BC_SMALLEST"';
    actual : STRING(500);
END_VAR
TEST('TestSerializeWith');

serializer.Reset();
_type.SerializeWith(serializer);
serializer.TryGetSerializedData(ADR(actual), SIZEOF(actual));

AssertEquals_STRING(
    Expected := expected,
    Actual := actual,
    Message := 'Serialization of type data did not return correct string.'
);

TEST_FINISHED();
END_METHOD

METHOD PUBLIC TestSize
VAR
    _type : _ETcVnBlobCombination(ETcVnBlobCombination.TCVN_BC_SMALLEST);
    expected : UDINT := SIZEOF(ETcVnBlobCombination);
    actual : UDINT;
END_VAR
TEST('TestSize');

actual := _type.Size;

AssertEquals_UDINT(
    Expected := Expected,
    Actual := actual,
    Message := 'Type did not return the correct size.'
);

TEST_FINISHED();
END_METHOD

METHOD PUBLIC TestTryDeserializeFrom
VAR
    deserializer : JsonDeserializer;
    feedback : DeserializerFeedback;
    json : STRING := '"TCVN_BC_SMALLEST"';
    _type : _ETcVnBlobCombination(ETcVnBlobCombination.TCVN_BC_SMALLEST);
    expected : ETcVnBlobCombination := ETcVnBlobCombination.TCVN_BC_SMALLEST;
    actual : ETcVnBlobCombination;
 END_VAR
TEST('TestTryDeserializeFrom');

deserializer.Reset();
deserializer.TryLoad(json);
_type.TryDeserializeFrom(Deserializer, Feedback);

actual := _type.Value;

AssertEquals(
    Expected := expected,
    Actual := actual,
    Message := 'Type did not deserialize correctly.'
);

TEST_FINISHED();
END_METHOD

METHOD PUBLIC TestTryMakeReferenceToFollowsReference
VAR
    _type : _ETcVnBlobCombination(ETcVnBlobCombination.TCVN_BC_SMALLEST);
	target : _ETcVnBlobCombination(ETcVnBlobCombination.TCVN_BC_SMALLEST);
    expected : ETcVnBlobCombination := ETcVnBlobCombination.TCVN_BC_LARGEST;
    actual : ETcVnBlobCombination;
END_VAR
TEST('TestTryMakeReferenceToFollowsReference');

_type.TryMakeReferenceTo(target);
target.Value := ETcVnBlobCombination.TCVN_BC_LARGEST;

actual := _type.Value;

AssertEquals(
    Expected := expected,
    Actual := actual,
    Message := 'Value did not follow target change.'
);

TEST_FINISHED();
END_METHOD

METHOD PUBLIC TestTryMakeReferenceToUpdatesReference
VAR
    _type : _ETcVnBlobCombination(ETcVnBlobCombination.TCVN_BC_SMALLEST);
	target : _ETcVnBlobCombination(ETcVnBlobCombination.TCVN_BC_SMALLEST);
    expected : ETcVnBlobCombination := ETcVnBlobCombination.TCVN_BC_LARGEST;
    actual : ETcVnBlobCombination;
END_VAR
TEST('TestTryMakeReferenceToUpdatesReference');

_type.TryMakeReferenceTo(target);
_type.Value := ETcVnBlobCombination.TCVN_BC_LARGEST;

actual := target.Value;

AssertEquals(
    Expected := expected,
    Actual := actual,
    Message := 'Value did not update target.'
);

TEST_FINISHED();
END_METHOD

METHOD PUBLIC TestTypeNameReturnsExpected
VAR
    _type : _ETcVnBlobCombination(ETcVnBlobCombination.TCVN_BC_SMALLEST);
    expected : STRING := 'ENUM';
    actual : STRING;
END_VAR
TEST('TestTypeNameReturnsExpected');

actual := _type.TypeName;

AssertEquals_STRING(
    Expected := expected,
    Actual := actual,
    Message := 'Type did not return correct iec type.'
);

TEST_FINISHED();
END_METHOD

METHOD PUBLIC TestValueReturnsExpectedAfterChange
VAR
    _type : _ETcVnBlobCombination(ETcVnBlobCombination.TCVN_BC_SMALLEST);
    expected : ETcVnBlobCombination := ETcVnBlobCombination.TCVN_BC_LARGEST;
    actual : ETcVnBlobCombination;
END_VAR
TEST('TestValueReturnsExpectedAfterChange');

_type.Value := ETcVnBlobCombination.TCVN_BC_LARGEST;

actual := _type.Value;

AssertEquals(
    Expected := expected,
    Actual := actual,
    Message := 'Expected value not returned after change.'
);

TEST_FINISHED();
END_METHOD

METHOD PUBLIC TestValueReturnsExpectedAfterInit
VAR
    _type : _ETcVnBlobCombination(ETcVnBlobCombination.TCVN_BC_SMALLEST);
    expected : ETcVnBlobCombination := ETcVnBlobCombination.TCVN_BC_SMALLEST;
    actual : ETcVnBlobCombination;
END_VAR
TEST('TestValueReturnsExpectedAfterInit');

actual := _type.Value;

AssertEquals(
    Expected := expected,
    Actual := actual,
    Message := 'Expected value not returned after Init.'
);

TEST_FINISHED();
END_METHOD

END_FUNCTION_BLOCK

// ---- Tests/Enums/_ETcVnBorderInterpolationMethod_TestSuite.TcPOU
FUNCTION_BLOCK _ETcVnBorderInterpolationMethod_TestSuite EXTENDS TcUnit.FB_TestSuite
VAR
END_VAR

TestAddress();
TestClearReference();
TestClone();
TestTypeNameReturnsExpected();
TestIdentifierReturnsExpected();
TestMakeReferenceToFollowsReference();
TestMakeReferenceToUpdatesReference();
TestSize();
TestValueReturnsExpectedAfterInit();
TestValueReturnsExpectedAfterChange();
TestSerializeTypeWith();
TestSerializeWith();
TestTryDeserializeFrom();
TestTryMakeReferenceToFollowsReference();
TestTryMakeReferenceToUpdatesReference();

METHOD PUBLIC TestAddress
VAR
    _type : _ETcVnBorderInterpolationMethod(ETcVnBorderInterpolationMethod.TCVN_BIM_CONSTANT);
    notExpected : PVOID := 0;
    actual : PVOID;
END_VAR
TEST('TestAddress');

actual := _type.Address;

AssertFalse(
    Condition := (notExpected = actual),
    Message := 'Type did not return a valid address.'
);

TEST_FINISHED();
END_METHOD

METHOD PUBLIC TestClearReference
VAR
    _type : _ETcVnBorderInterpolationMethod(ETcVnBorderInterpolationMethod.TCVN_BIM_CONSTANT);
	target : ETcVnBorderInterpolationMethod := ETcVnBorderInterpolationMethod.TCVN_BIM_CONSTANT;
    expected : ETcVnBorderInterpolationMethod := ETcVnBorderInterpolationMethod.TCVN_BIM_CONSTANT;
    actual : ETcVnBorderInterpolationMethod;
END_VAR
TEST('TestClearReference');

_type.MakeReferenceTo(target);
_type.ClearReference();
target := ETcVnBorderInterpolationMethod.TCVN_BIM_REPLICATE;

actual := _type.Value;

AssertEquals(
    Expected := expected,
    Actual := actual,
    Message := 'Value continued to follow target.'
);

TEST_FINISHED();
END_METHOD

METHOD PUBLIC TestClone
VAR
    _type : _ETcVnBorderInterpolationMethod(ETcVnBorderInterpolationMethod.TCVN_BIM_CONSTANT);
	clone : I_Datatype;
	isValidClone : BOOL;
	compareResult : DINT;
END_VAR
TEST('TestClone');

clone := _type.Clone();

isValidClone := clone <> 0;

IF isValidClone THEN
	compareResult := memcmp(_type.Address, clone.Address, clone.Size);
END_IF

AssertTrue(
	Condition := isValidClone,
	Message := 'Clone did not produce a clone'
);

AssertEquals_DINT(
	Expected := 0,
    Actual := compareResult,
    Message := 'Clone did not return a valid clone.'
);

clone.Dispose();

TEST_FINISHED();
END_METHOD

METHOD PUBLIC TestIdentifierReturnsExpected
VAR
    _type : _ETcVnBorderInterpolationMethod(ETcVnBorderInterpolationMethod.TCVN_BIM_CONSTANT);
    expected : STRING := 'ETcVnBorderInterpolationMethod';
    actual : STRING;
END_VAR
TEST('TestIdentifierReturnsExpected');

actual := _type.Identifier;

AssertEquals_STRING(
    Expected := expected,
    Actual := actual,
    Message := 'Type did not return correct iec type.'
);

TEST_FINISHED();
END_METHOD

METHOD PUBLIC TestMakeReferenceToFollowsReference
VAR
    _type : _ETcVnBorderInterpolationMethod(ETcVnBorderInterpolationMethod.TCVN_BIM_CONSTANT);
	target : ETcVnBorderInterpolationMethod := ETcVnBorderInterpolationMethod.TCVN_BIM_CONSTANT;
    expected : ETcVnBorderInterpolationMethod := ETcVnBorderInterpolationMethod.TCVN_BIM_REPLICATE;
    actual : ETcVnBorderInterpolationMethod;
END_VAR
TEST('TestMakeReferenceToFollowsReference');

_type.MakeReferenceTo(target);
target := ETcVnBorderInterpolationMethod.TCVN_BIM_REPLICATE;

actual := _type.Value;

AssertEquals(
    Expected := expected,
    Actual := actual,
    Message := 'Value did not follow target change.'
);

TEST_FINISHED();
END_METHOD

METHOD PUBLIC TestMakeReferenceToUpdatesReference
VAR
    _type : _ETcVnBorderInterpolationMethod(ETcVnBorderInterpolationMethod.TCVN_BIM_CONSTANT);
	target : ETcVnBorderInterpolationMethod := ETcVnBorderInterpolationMethod.TCVN_BIM_CONSTANT;
    expected : ETcVnBorderInterpolationMethod := ETcVnBorderInterpolationMethod.TCVN_BIM_REPLICATE;
    actual : ETcVnBorderInterpolationMethod;
END_VAR
TEST('TestMakeReferenceToUpdatesReference');

_type.MakeReferenceTo(target);
_type.Value := ETcVnBorderInterpolationMethod.TCVN_BIM_REPLICATE;

actual := target;

AssertEquals(
    Expected := expected,
    Actual := actual,
    Message := 'Value did not update target.'
);

TEST_FINISHED();
END_METHOD

METHOD PUBLIC TestSerializeTypeWith
VAR
    _type : _ETcVnBorderInterpolationMethod(ETcVnBorderInterpolationMethod.TCVN_BIM_CONSTANT);
    serializer : JsonSerializer;
    expected : STRING(500) := '{"typeName":"ENUM","identifier":"ETcVnBorderInterpolationMethod","enumerations":["TCVN_BIM_CONSTANT","TCVN_BIM_REPLICATE","TCVN_BIM_REFLECT","TCVN_BIM_WRAP","TCVN_BIM_REFLECT_101","TCVN_BIM_DEFAULT","TCVN_BIM_TRANSPARENT","TCVN_BIM_ISOLATED_CONSTANT","TCVN_BIM_ISOLATED_REPLICATE","TCVN_BIM_ISOLATED_REFLECT","TCVN_BIM_ISOLATED_WRAP","TCVN_BIM_ISOLATED_REFLECT_101"],"baseType":{"typeName":"DINT","minValue":-2147483648,"maxValue":2147483647,"isSigned":true,"isFloat":false}}'; 
    actual : STRING(500);
END_VAR
TEST('TestSerializeTypeWith');

serializer.Reset();
_type.SerializeTypeWith(serializer);
serializer.TryGetSerializedData(ADR(actual), SIZEOF(actual));

AssertEquals_STRING(
    Expected := expected,
    Actual := actual,
    Message := 'Serialization of type did not return correct string.'
);

TEST_FINISHED();
END_METHOD

METHOD PUBLIC TestSerializeWith
VAR
    _type : _ETcVnBorderInterpolationMethod(ETcVnBorderInterpolationMethod.TCVN_BIM_CONSTANT);
    serializer : JsonSerializer;
    expected : STRING := '"TCVN_BIM_CONSTANT"';
    actual : STRING(500);
END_VAR
TEST('TestSerializeWith');

serializer.Reset();
_type.SerializeWith(serializer);
serializer.TryGetSerializedData(ADR(actual), SIZEOF(actual));

AssertEquals_STRING(
    Expected := expected,
    Actual := actual,
    Message := 'Serialization of type data did not return correct string.'
);

TEST_FINISHED();
END_METHOD

METHOD PUBLIC TestSize
VAR
    _type : _ETcVnBorderInterpolationMethod(ETcVnBorderInterpolationMethod.TCVN_BIM_CONSTANT);
    expected : UDINT := SIZEOF(ETcVnBorderInterpolationMethod);
    actual : UDINT;
END_VAR
TEST('TestSize');

actual := _type.Size;

AssertEquals_UDINT(
    Expected := Expected,
    Actual := actual,
    Message := 'Type did not return the correct size.'
);

TEST_FINISHED();
END_METHOD

METHOD PUBLIC TestTryDeserializeFrom
VAR
    deserializer : JsonDeserializer;
    feedback : DeserializerFeedback;
    json : STRING := '"TCVN_BIM_CONSTANT"';
    _type : _ETcVnBorderInterpolationMethod(ETcVnBorderInterpolationMethod.TCVN_BIM_CONSTANT);
    expected : ETcVnBorderInterpolationMethod := ETcVnBorderInterpolationMethod.TCVN_BIM_CONSTANT;
    actual : ETcVnBorderInterpolationMethod;
 END_VAR
TEST('TestTryDeserializeFrom');

deserializer.Reset();
deserializer.TryLoad(json);
_type.TryDeserializeFrom(Deserializer, Feedback);

actual := _type.Value;

AssertEquals(
    Expected := expected,
    Actual := actual,
    Message := 'Type did not deserialize correctly.'
);

TEST_FINISHED();
END_METHOD

METHOD PUBLIC TestTryMakeReferenceToFollowsReference
VAR
    _type : _ETcVnBorderInterpolationMethod(ETcVnBorderInterpolationMethod.TCVN_BIM_CONSTANT);
	target : _ETcVnBorderInterpolationMethod(ETcVnBorderInterpolationMethod.TCVN_BIM_CONSTANT);
    expected : ETcVnBorderInterpolationMethod := ETcVnBorderInterpolationMethod.TCVN_BIM_REPLICATE;
    actual : ETcVnBorderInterpolationMethod;
END_VAR
TEST('TestTryMakeReferenceToFollowsReference');

_type.TryMakeReferenceTo(target);
target.Value := ETcVnBorderInterpolationMethod.TCVN_BIM_REPLICATE;

actual := _type.Value;

AssertEquals(
    Expected := expected,
    Actual := actual,
    Message := 'Value did not follow target change.'
);

TEST_FINISHED();
END_METHOD

METHOD PUBLIC TestTryMakeReferenceToUpdatesReference
VAR
    _type : _ETcVnBorderInterpolationMethod(ETcVnBorderInterpolationMethod.TCVN_BIM_CONSTANT);
	target : _ETcVnBorderInterpolationMethod(ETcVnBorderInterpolationMethod.TCVN_BIM_CONSTANT);
    expected : ETcVnBorderInterpolationMethod := ETcVnBorderInterpolationMethod.TCVN_BIM_REPLICATE;
    actual : ETcVnBorderInterpolationMethod;
END_VAR
TEST('TestTryMakeReferenceToUpdatesReference');

_type.TryMakeReferenceTo(target);
_type.Value := ETcVnBorderInterpolationMethod.TCVN_BIM_REPLICATE;

actual := target.Value;

AssertEquals(
    Expected := expected,
    Actual := actual,
    Message := 'Value did not update target.'
);

TEST_FINISHED();
END_METHOD

METHOD PUBLIC TestTypeNameReturnsExpected
VAR
    _type : _ETcVnBorderInterpolationMethod(ETcVnBorderInterpolationMethod.TCVN_BIM_CONSTANT);
    expected : STRING := 'ENUM';
    actual : STRING;
END_VAR
TEST('TestTypeNameReturnsExpected');

actual := _type.TypeName;

AssertEquals_STRING(
    Expected := expected,
    Actual := actual,
    Message := 'Type did not return correct iec type.'
);

TEST_FINISHED();
END_METHOD

METHOD PUBLIC TestValueReturnsExpectedAfterChange
VAR
    _type : _ETcVnBorderInterpolationMethod(ETcVnBorderInterpolationMethod.TCVN_BIM_CONSTANT);
    expected : ETcVnBorderInterpolationMethod := ETcVnBorderInterpolationMethod.TCVN_BIM_REPLICATE;
    actual : ETcVnBorderInterpolationMethod;
END_VAR
TEST('TestValueReturnsExpectedAfterChange');

_type.Value := ETcVnBorderInterpolationMethod.TCVN_BIM_REPLICATE;

actual := _type.Value;

AssertEquals(
    Expected := expected,
    Actual := actual,
    Message := 'Expected value not returned after change.'
);

TEST_FINISHED();
END_METHOD

METHOD PUBLIC TestValueReturnsExpectedAfterInit
VAR
    _type : _ETcVnBorderInterpolationMethod(ETcVnBorderInterpolationMethod.TCVN_BIM_CONSTANT);
    expected : ETcVnBorderInterpolationMethod := ETcVnBorderInterpolationMethod.TCVN_BIM_CONSTANT;
    actual : ETcVnBorderInterpolationMethod;
END_VAR
TEST('TestValueReturnsExpectedAfterInit');

actual := _type.Value;

AssertEquals(
    Expected := expected,
    Actual := actual,
    Message := 'Expected value not returned after Init.'
);

TEST_FINISHED();
END_METHOD

END_FUNCTION_BLOCK

// ---- Tests/Enums/_ETcVnColorSpaceTransform_TestSuite.TcPOU
FUNCTION_BLOCK _ETcVnColorSpaceTransform_TestSuite EXTENDS TcUnit.FB_TestSuite
VAR
END_VAR

TestAddress();
TestClearReference();
TestClone();
TestTypeNameReturnsExpected();
TestIdentifierReturnsExpected();
TestMakeReferenceToFollowsReference();
TestMakeReferenceToUpdatesReference();
TestSize();
TestValueReturnsExpectedAfterInit();
TestValueReturnsExpectedAfterChange();
TestSerializeTypeWith();
TestSerializeWith();
TestTryDeserializeFrom();
TestTryMakeReferenceToFollowsReference();
TestTryMakeReferenceToUpdatesReference();

METHOD PUBLIC TestAddress
VAR
    _type : _ETcVnColorSpaceTransform(ETcVnColorSpaceTransform.TCVN_CST_BGR_TO_BGRA);
    notExpected : PVOID := 0;
    actual : PVOID;
END_VAR
TEST('TestAddress');

actual := _type.Address;

AssertFalse(
    Condition := (notExpected = actual),
    Message := 'Type did not return a valid address.'
);

TEST_FINISHED();
END_METHOD

METHOD PUBLIC TestClearReference
VAR
    _type : _ETcVnColorSpaceTransform(ETcVnColorSpaceTransform.TCVN_CST_BGR_TO_BGRA);
	target : ETcVnColorSpaceTransform := ETcVnColorSpaceTransform.TCVN_CST_BGR_TO_BGRA;
    expected : ETcVnColorSpaceTransform := ETcVnColorSpaceTransform.TCVN_CST_BGR_TO_BGRA;
    actual : ETcVnColorSpaceTransform;
END_VAR
TEST('TestClearReference');

_type.MakeReferenceTo(target);
_type.ClearReference();
target := ETcVnColorSpaceTransform.TCVN_CST_MAX;

actual := _type.Value;

AssertEquals(
    Expected := expected,
    Actual := actual,
    Message := 'Value continued to follow target.'
);

TEST_FINISHED();
END_METHOD

METHOD PUBLIC TestClone
VAR
    _type : _ETcVnColorSpaceTransform(ETcVnColorSpaceTransform.TCVN_CST_BGR_TO_BGRA);
	clone : I_Datatype;
	isValidClone : BOOL;
	compareResult : DINT;
END_VAR
TEST('TestClone');

clone := _type.Clone();

isValidClone := clone <> 0;

IF isValidClone THEN
	compareResult := memcmp(_type.Address, clone.Address, clone.Size);
END_IF

AssertTrue(
	Condition := isValidClone,
	Message := 'Clone did not produce a clone'
);

AssertEquals_DINT(
	Expected := 0,
    Actual := compareResult,
    Message := 'Clone did not return a valid clone.'
);

clone.Dispose();

TEST_FINISHED();
END_METHOD

METHOD PUBLIC TestIdentifierReturnsExpected
VAR
    _type : _ETcVnColorSpaceTransform(ETcVnColorSpaceTransform.TCVN_CST_BGR_TO_BGRA);
    expected : STRING := 'ETcVnColorSpaceTransform';
    actual : STRING;
END_VAR
TEST('TestIdentifierReturnsExpected');

actual := _type.Identifier;

AssertEquals_STRING(
    Expected := expected,
    Actual := actual,
    Message := 'Type did not return correct iec type.'
);

TEST_FINISHED();
END_METHOD

METHOD PUBLIC TestMakeReferenceToFollowsReference
VAR
    _type : _ETcVnColorSpaceTransform(ETcVnColorSpaceTransform.TCVN_CST_BGR_TO_BGRA);
	target : ETcVnColorSpaceTransform := ETcVnColorSpaceTransform.TCVN_CST_BGR_TO_BGRA;
    expected : ETcVnColorSpaceTransform := ETcVnColorSpaceTransform.TCVN_CST_MAX;
    actual : ETcVnColorSpaceTransform;
END_VAR
TEST('TestMakeReferenceToFollowsReference');

_type.MakeReferenceTo(target);
target := ETcVnColorSpaceTransform.TCVN_CST_MAX;

actual := _type.Value;

AssertEquals(
    Expected := expected,
    Actual := actual,
    Message := 'Value did not follow target change.'
);

TEST_FINISHED();
END_METHOD

METHOD PUBLIC TestMakeReferenceToUpdatesReference
VAR
    _type : _ETcVnColorSpaceTransform(ETcVnColorSpaceTransform.TCVN_CST_BGR_TO_BGRA);
	target : ETcVnColorSpaceTransform := ETcVnColorSpaceTransform.TCVN_CST_BGR_TO_BGRA;
    expected : ETcVnColorSpaceTransform := ETcVnColorSpaceTransform.TCVN_CST_MAX;
    actual : ETcVnColorSpaceTransform;
END_VAR
TEST('TestMakeReferenceToUpdatesReference');

_type.MakeReferenceTo(target);
_type.Value := ETcVnColorSpaceTransform.TCVN_CST_MAX;

actual := target;

AssertEquals(
    Expected := expected,
    Actual := actual,
    Message := 'Value did not update target.'
);

TEST_FINISHED();
END_METHOD

METHOD PUBLIC TestSerializeTypeWith
VAR
    _type : _ETcVnColorSpaceTransform(ETcVnColorSpaceTransform.TCVN_CST_BGR_TO_BGRA);
    serializer : JsonSerializer;
    expected : STRING(6000) := '{"typeName":"ENUM","identifier":"ETcVnColorSpaceTransform","enumerations":["TCVN_CST_BGR_TO_BGRA","TCVN_CST_RGB_TO_RGBA","TCVN_CST_BGRA_TO_BGR","TCVN_CST_RGBA_TO_RGB","TCVN_CST_BGR_TO_RGBA","TCVN_CST_RGB_TO_BGRA","TCVN_CST_BGRA_TO_RGB","TCVN_CST_RGBA_TO_BGR","TCVN_CST_BGR_TO_RGB","TCVN_CST_RGB_TO_BGR","TCVN_CST_BGRA_TO_RGBA","TCVN_CST_RGBA_TO_BGRA","TCVN_CST_BGR_TO_GRAY","TCVN_CST_RGB_TO_GRAY","TCVN_CST_GRAY_TO_BGR","TCVN_CST_GRAY_TO_RGB","TCVN_CST_GRAY_TO_BGRA","TCVN_CST_GRAY_TO_RGBA","TCVN_CST_BGRA_TO_GRAY","TCVN_CST_RGBA_TO_GRAY","TCVN_CST_RGB_TO_BGR_565","TCVN_CST_BGR_TO_BGR_565","TCVN_CST_BGR_565_TO_RGB","TCVN_CST_BGR_565_TO_BGR","TCVN_CST_RGBA_TO_BGR_565","TCVN_CST_BGRA_TO_BGR_565","TCVN_CST_BGR_565_TO_RGBA","TCVN_CST_BGR_565_TO_BGRA","TCVN_CST_GRAY_TO_BGR_565","TCVN_CST_BGR_565_TO_GRAY","TCVN_CST_RGB_TO_BGR_555","TCVN_CST_BGR_TO_BGR_555","TCVN_CST_BGR_555_TO_RGB","TCVN_CST_BGR_555_TO_BGR","TCVN_CST_RGBA_TO_BGR_555","TCVN_CST_BGRA_TO_BGR_555","TCVN_CST_BGR_555_TO_RGBA","TCVN_CST_BGR_555_TO_BGRA","TCVN_CST_GRAY_TO_BGR_555","TCVN_CST_BGR_555_TO_GRAY","TCVN_CST_BGR_TO_XYZ","TCVN_CST_RGB_TO_XYZ","TCVN_CST_XYZ_TO_BGR","TCVN_CST_XYZ_TO_RGB","TCVN_CST_BGR_TO_YCRCB","TCVN_CST_RGB_TO_YCRCB","TCVN_CST_YCRCB_TO_BGR","TCVN_CST_YCRCB_TO_RGB","TCVN_CST_BGR_TO_HSV","TCVN_CST_RGB_TO_HSV","TCVN_CST_BGR_TO_LAB","TCVN_CST_RGB_TO_LAB","TCVN_CST_BAYER_RG_TO_BGR","TCVN_CST_BAYER_BG_TO_RGB","TCVN_CST_BAYER_GR_TO_BGR","TCVN_CST_BAYER_GB_TO_RGB","TCVN_CST_BAYER_BG_TO_BGR","TCVN_CST_BAYER_RG_TO_RGB","TCVN_CST_BAYER_GB_TO_BGR","TCVN_CST_BAYER_GR_TO_RGB","TCVN_CST_BGR_TO_LUV","TCVN_CST_RGB_TO_LUV","TCVN_CST_BGR_TO_HLS","TCVN_CST_RGB_TO_HLS","TCVN_CST_HSV_TO_BGR","TCVN_CST_HSV_TO_RGB","TCVN_CST_LAB_TO_BGR","TCVN_CST_LAB_TO_RGB","TCVN_CST_LUV_TO_BGR","TCVN_CST_LUV_TO_RGB","TCVN_CST_HLS_TO_BGR","TCVN_CST_HLS_TO_RGB","TCVN_CST_BAYER_RG_TO_BGR_VNG","TCVN_CST_BAYER_GR_TO_BGR_VNG","TCVN_CST_BAYER_BG_TO_BGR_VNG","TCVN_CST_BAYER_GB_TO_BGR_VNG","TCVN_CST_BAYER_RG_TO_RGB_VNG","TCVN_CST_BAYER_GR_TO_RGB_VNG","TCVN_CST_BAYER_BG_TO_RGB_VNG","TCVN_CST_BAYER_GB_TO_RGB_VNG","TCVN_CST_BGR_TO_HSV_FULL","TCVN_CST_RGB_TO_HSV_FULL","TCVN_CST_BGR_TO_HLS_FULL","TCVN_CST_RGB_TO_HLS_FULL","TCVN_CST_HSV_TO_BGR_FULL","TCVN_CST_HSV_TO_RGB_FULL","TCVN_CST_HLS_TO_BGR_FULL","TCVN_CST_HLS_TO_RGB_FULL","TCVN_CST_LBGR_TO_LAB","TCVN_CST_LRGB_TO_LAB","TCVN_CST_LBGR_TO_LUV","TCVN_CST_LRGB_TO_LUV","TCVN_CST_LAB_TO_LBGR","TCVN_CST_LAB_TO_LRGB","TCVN_CST_LUV_TO_LBGR","TCVN_CST_LUV_TO_LRGB","TCVN_CST_BGR_TO_YUV","TCVN_CST_RGB_TO_YUV","TCVN_CST_YUV_TO_BGR","TCVN_CST_YUV_TO_RGB","TCVN_CST_BAYER_RG_TO_GRAY","TCVN_CST_BAYER_GR_TO_GRAY","TCVN_CST_BAYER_BG_TO_GRAY","TCVN_CST_BAYER_GB_TO_GRAY","TCVN_CST_YUV_420_NV12_TO_RGB","TCVN_CST_YUV_420_NV12_TO_BGR","TCVN_CST_YUV_420_NV21_TO_RGB","TCVN_CST_YUV_420_NV21_TO_BGR","TCVN_CST_YUV_420_SP_TO_RGB","TCVN_CST_YUV_420_SP_TO_BGR","TCVN_CST_YUV_420_NV12_TO_RGBA","TCVN_CST_YUV_420_NV12_TO_BGRA","TCVN_CST_YUV_420_NV21_TO_RGBA","TCVN_CST_YUV_420_NV21_TO_BGRA","TCVN_CST_YUV_420_SP_TO_RGBA","TCVN_CST_YUV_420_SP_TO_BGRA","TCVN_CST_YUV_420_YV12_TO_RGB","TCVN_CST_YUV_420_YV12_TO_BGR","TCVN_CST_YUV_420_IYUV_TO_RGB","TCVN_CST_YUV_420_IYUV_TO_BGR","TCVN_CST_YUV_420_I420_TO_RGB","TCVN_CST_YUV_420_I420_TO_BGR","TCVN_CST_YUV_420_P_TO_RGB","TCVN_CST_YUV_420_P_TO_BGR","TCVN_CST_YUV_420_YV12_TO_RGBA","TCVN_CST_YUV_420_YV12_TO_BGRA","TCVN_CST_YUV_420_IYUV_TO_RGBA","TCVN_CST_YUV_420_IYUV_TO_BGRA","TCVN_CST_YUV_420_I420_TO_RGBA","TCVN_CST_YUV_420_I420_TO_BGRA","TCVN_CST_YUV_420_P_TO_RGBA","TCVN_CST_YUV_420_P_TO_BGRA","TCVN_CST_YUV_420_TO_GRAY","TCVN_CST_YUV_420_NV21_TO_GRAY","TCVN_CST_YUV_420_NV12_TO_GRAY","TCVN_CST_YUV_420_YV12_TO_GRAY","TCVN_CST_YUV_420_IYUV_TO_GRAY","TCVN_CST_YUV_420_I420_TO_GRAY","TCVN_CST_YUV_420_SP_TO_GRAY","TCVN_CST_YUV_420_P_TO_GRAY","TCVN_CST_YUV_422_UYVY_TO_RGB","TCVN_CST_YUV_422_UYVY_TO_BGR","TCVN_CST_YUV_422_Y422_TO_RGB","TCVN_CST_YUV_422_Y422_TO_BGR","TCVN_CST_YUV_422_UYNV_TO_RGB","TCVN_CST_YUV_422_UYNV_TO_BGR","TCVN_CST_YUV_422_UYVY_TO_RGBA","TCVN_CST_YUV_422_UYVY_TO_BGRA","TCVN_CST_YUV_422_Y422_TO_RGBA","TCVN_CST_YUV_422_Y422_TO_BGRA","TCVN_CST_YUV_422_UYNV_TO_RGBA","TCVN_CST_YUV_422_UYNV_TO_BGRA","TCVN_CST_YUV_422_YUY2_TO_RGB","TCVN_CST_YUV_422_YUY2_TO_BGR","TCVN_CST_YUV_422_YVYU_TO_RGB","TCVN_CST_YUV_422_YVYU_TO_BGR","TCVN_CST_YUV_422_YUYV_TO_RGB","TCVN_CST_YUV_422_YUYV_TO_BGR","TCVN_CST_YUV_422_YUNV_TO_RGB","TCVN_CST_YUV_422_YUNV_TO_BGR","TCVN_CST_YUV_422_YUY2_TO_RGBA","TCVN_CST_YUV_422_YUY2_TO_BGRA","TCVN_CST_YUV_422_YVYU_TO_RGBA","TCVN_CST_YUV_422_YVYU_TO_BGRA","TCVN_CST_YUV_422_YUYV_TO_RGBA","TCVN_CST_YUV_422_YUYV_TO_BGRA","TCVN_CST_YUV_422_YUNV_TO_RGBA","TCVN_CST_YUV_422_YUNV_TO_BGRA","TCVN_CST_YUV_422_UYVY_TO_GRAY","TCVN_CST_YUV_422_YUY2_TO_GRAY","TCVN_CST_YUV_422_Y422_TO_GRAY","TCVN_CST_YUV_422_UYNV_TO_GRAY","TCVN_CST_YUV_422_YVYU_TO_GRAY","TCVN_CST_YUV_422_YUYV_TO_GRAY","TCVN_CST_YUV_422_YUNV_TO_GRAY","TCVN_CST_RGBA_TO_PREMULTIPLICATED_RGBA","TCVN_CST_PREMULTIPLICATED_RGBA_TO_RGBA","TCVN_CST_RGB_TO_YUV_420_I420","TCVN_CST_BGR_TO_YUV_420_I420","TCVN_CST_RGB_TO_YUV_420_IYUV","TCVN_CST_BGR_TO_YUV_420_IYUV","TCVN_CST_RGBA_TO_YUV_420_I420","TCVN_CST_BGRA_TO_YUV_420_I420","TCVN_CST_RGBA_TO_YUV_420_IYUV","TCVN_CST_BGRA_TO_YUV_420_IYUV","TCVN_CST_RGB_TO_YUV_420_YV12","TCVN_CST_BGR_TO_YUV_420_YV12","TCVN_CST_RGBA_TO_YUV_420_YV12","TCVN_CST_BGRA_TO_YUV_420_YV12","TCVN_CST_BAYER_RG_TO_BGR_EA","TCVN_CST_BAYER_GR_TO_BGR_EA","TCVN_CST_BAYER_BG_TO_BGR_EA","TCVN_CST_BAYER_GB_TO_BGR_EA","TCVN_CST_BAYER_RG_TO_RGB_EA","TCVN_CST_BAYER_GR_TO_RGB_EA","TCVN_CST_BAYER_BG_TO_RGB_EA","TCVN_CST_BAYER_GB_TO_RGB_EA","TCVN_CST_BAYER_RG_TO_BGRA","TCVN_CST_BAYER_GR_TO_BGRA","TCVN_CST_BAYER_BG_TO_BGRA","TCVN_CST_BAYER_GB_TO_BGRA","TCVN_CST_BAYER_RG_TO_RGBA","TCVN_CST_BAYER_GR_TO_RGBA","TCVN_CST_BAYER_BG_TO_RGBA","TCVN_CST_BAYER_GB_TO_RGBA","TCVN_CST_MAX"],"baseType":{"typeName":"DINT","minValue":-2147483648,"maxValue":2147483647,"isSigned":true,"isFloat":false}}'; 
    actual : STRING(6000);
END_VAR
TEST('TestSerializeTypeWith');

serializer.Reset();
_type.SerializeTypeWith(serializer);
serializer.TryGetSerializedData(ADR(actual), SIZEOF(actual));

AssertEquals_STRING(
    Expected := expected,
    Actual := actual,
    Message := 'Serialization of type did not return correct string.'
);

TEST_FINISHED();
END_METHOD

METHOD PUBLIC TestSerializeWith
VAR
    _type : _ETcVnColorSpaceTransform(ETcVnColorSpaceTransform.TCVN_CST_BGR_TO_BGRA);
    serializer : JsonSerializer;
    expected : STRING := '"TCVN_CST_BGR_TO_BGRA"';
    actual : STRING(500);
END_VAR
TEST('TestSerializeWith');

serializer.Reset();
_type.SerializeWith(serializer);
serializer.TryGetSerializedData(ADR(actual), SIZEOF(actual));

AssertEquals_STRING(
    Expected := expected,
    Actual := actual,
    Message := 'Serialization of type data did not return correct string.'
);

TEST_FINISHED();
END_METHOD

METHOD PUBLIC TestSize
VAR
    _type : _ETcVnColorSpaceTransform(ETcVnColorSpaceTransform.TCVN_CST_BGR_TO_BGRA);
    expected : UDINT := SIZEOF(ETcVnColorSpaceTransform);
    actual : UDINT;
END_VAR
TEST('TestSize');

actual := _type.Size;

AssertEquals_UDINT(
    Expected := Expected,
    Actual := actual,
    Message := 'Type did not return the correct size.'
);

TEST_FINISHED();
END_METHOD

METHOD PUBLIC TestTryDeserializeFrom
VAR
    deserializer : JsonDeserializer;
    feedback : DeserializerFeedback;
    json : STRING := '"TCVN_CST_BGR_TO_BGRA"';
    _type : _ETcVnColorSpaceTransform(ETcVnColorSpaceTransform.TCVN_CST_BGR_TO_BGRA);
    expected : ETcVnColorSpaceTransform := ETcVnColorSpaceTransform.TCVN_CST_BGR_TO_BGRA;
    actual : ETcVnColorSpaceTransform;
 END_VAR
TEST('TestTryDeserializeFrom');

deserializer.Reset();
deserializer.TryLoad(json);
_type.TryDeserializeFrom(Deserializer, Feedback);

actual := _type.Value;

AssertEquals(
    Expected := expected,
    Actual := actual,
    Message := 'Type did not deserialize correctly.'
);

TEST_FINISHED();
END_METHOD

METHOD PUBLIC TestTryMakeReferenceToFollowsReference
VAR
    _type : _ETcVnColorSpaceTransform(ETcVnColorSpaceTransform.TCVN_CST_BGR_TO_BGRA);
	target : _ETcVnColorSpaceTransform(ETcVnColorSpaceTransform.TCVN_CST_BGR_TO_BGRA);
    expected : ETcVnColorSpaceTransform := ETcVnColorSpaceTransform.TCVN_CST_MAX;
    actual : ETcVnColorSpaceTransform;
END_VAR
TEST('TestTryMakeReferenceToFollowsReference');

_type.TryMakeReferenceTo(target);
target.Value := ETcVnColorSpaceTransform.TCVN_CST_MAX;

actual := _type.Value;

AssertEquals(
    Expected := expected,
    Actual := actual,
    Message := 'Value did not follow target change.'
);

TEST_FINISHED();
END_METHOD

METHOD PUBLIC TestTryMakeReferenceToUpdatesReference
VAR
    _type : _ETcVnColorSpaceTransform(ETcVnColorSpaceTransform.TCVN_CST_BGR_TO_BGRA);
	target : _ETcVnColorSpaceTransform(ETcVnColorSpaceTransform.TCVN_CST_BGR_TO_BGRA);
    expected : ETcVnColorSpaceTransform := ETcVnColorSpaceTransform.TCVN_CST_MAX;
    actual : ETcVnColorSpaceTransform;
END_VAR
TEST('TestTryMakeReferenceToUpdatesReference');

_type.TryMakeReferenceTo(target);
_type.Value := ETcVnColorSpaceTransform.TCVN_CST_MAX;

actual := target.Value;

AssertEquals(
    Expected := expected,
    Actual := actual,
    Message := 'Value did not update target.'
);

TEST_FINISHED();
END_METHOD

METHOD PUBLIC TestTypeNameReturnsExpected
VAR
    _type : _ETcVnColorSpaceTransform(ETcVnColorSpaceTransform.TCVN_CST_BGR_TO_BGRA);
    expected : STRING := 'ENUM';
    actual : STRING;
END_VAR
TEST('TestTypeNameReturnsExpected');

actual := _type.TypeName;

AssertEquals_STRING(
    Expected := expected,
    Actual := actual,
    Message := 'Type did not return correct iec type.'
);

TEST_FINISHED();
END_METHOD

METHOD PUBLIC TestValueReturnsExpectedAfterChange
VAR
    _type : _ETcVnColorSpaceTransform(ETcVnColorSpaceTransform.TCVN_CST_BGR_TO_BGRA);
    expected : ETcVnColorSpaceTransform := ETcVnColorSpaceTransform.TCVN_CST_MAX;
    actual : ETcVnColorSpaceTransform;
END_VAR
TEST('TestValueReturnsExpectedAfterChange');

_type.Value := ETcVnColorSpaceTransform.TCVN_CST_MAX;

actual := _type.Value;

AssertEquals(
    Expected := expected,
    Actual := actual,
    Message := 'Expected value not returned after change.'
);

TEST_FINISHED();
END_METHOD

METHOD PUBLIC TestValueReturnsExpectedAfterInit
VAR
    _type : _ETcVnColorSpaceTransform(ETcVnColorSpaceTransform.TCVN_CST_BGR_TO_BGRA);
    expected : ETcVnColorSpaceTransform := ETcVnColorSpaceTransform.TCVN_CST_BGR_TO_BGRA;
    actual : ETcVnColorSpaceTransform;
END_VAR
TEST('TestValueReturnsExpectedAfterInit');

actual := _type.Value;

AssertEquals(
    Expected := expected,
    Actual := actual,
    Message := 'Expected value not returned after Init.'
);

TEST_FINISHED();
END_METHOD

END_FUNCTION_BLOCK
